      A     #Day6;  // Day 6 (Saturday)
      JNB   ED6;
      L     #EveningDay1Value;  // amount of bodies on day 1 - Evening shift (Monday)
      L     #EveningDay2Value;  // amount of bodies on day 2 - Evening shift (Tuesday)
      +I;
      L     #EveningDay3Value;  // amount of bodies on day 3 - Evening shift (Wednesday)
      +I;
      L     #EveningDay4Value;  // amount of bodies on day 4 - Evening shift (Thursday)
      +I;
      L     #EveningDay5Value;  // amount of bodies on day 5 - Evening shift (Friday)
      +I;
      L     #EveningDay6Value;  // amount of bodies on day 6 - Evening shift (Saturday)
      +I;
      T     #H_Out.TotalEvening;  // copy to HMI
ED6:  NOP   0;

      A     #Day7;  // Day 7 (Sunday)
      JNB   ED7;
      L     #EveningDay1Value;  // amount of bodies on day 1 - Evening shift (Monday)
      L     #EveningDay2Value;  // amount of bodies on day 2 - Evening shift (Tuesday)
      +I;
      L     #EveningDay3Value;  // amount of bodies on day 3 - Evening shift (Wednesday)
      +I;
      L     #EveningDay4Value;  // amount of bodies on day 4 - Evening shift (Thursday)
      +I;
      L     #EveningDay5Value;  // amount of bodies on day 5 - Evening shift (Friday)
      +I;
      L     #EveningDay6Value;  // amount of bodies on day 6 - Evening shift (Saturday)
      +I;
      L     #EveningDay7Value;  // amount of bodies on day 7 - Evening shift (Sunday)
      +I;
      T     #H_Out.TotalEvening;  // copy to HMI
ED7:  NOP   0;


NETWORK
TITLE = **** 4.4 - Machine status - Calculated **** Production value Night shift
// Production value Night shift
      A     #Day1;  // Day 1 (Monday)
      JNB   ND1;
      L     #NightDay1Value;  // amount of bodies on day 1 - Night shift (Monday)
      T     #H_Out.TotalNight;  // copy to HMI
ND1:  NOP   0;

      A     #Day2;  // Day 2 (tuesday)
      JNB   ND2;
      L     #NightDay1Value;  // amount of bodies on day 1 - Night shift (Monday)
      L     #NightDay2Value;  // amount of bodies on day 2 - Night shift (Tuesday)
      T     #H_Out.TotalNight;  // copy to HMI
ND2:  NOP   0;

      A     #Day3;  // Day 3 (Wednesday)
      JNB   ND3;
      L     #NightDay1Value;  // amount of bodies on day 1 - Night shift (Monday)
      L     #NightDay2Value;  // amount of bodies on day 2 - Night shift (Tuesday)
      +I;
      L     #NightDay3Value;  // amount of bodies on day 3 - Night shift (Wednesday)
      +I;
      T     #H_Out.TotalNight;  // copy to HMI
ND3:  NOP   0;

      A     #Day4;  // Day 4 (tuesday)
      JNB   ND4;
      L     #NightDay1Value;  // amount of bodies on day 1 - Night shift (Monday)
      L     #NightDay2Value;  // amount of bodies on day 2 - Night shift (Tuesday)
      +I;
      L     #NightDay3Value;  // amount of bodies on day 3 - Night shift (Wednesday)
      +I;
      L     #NightDay4Value;  // amount of bodies on day 4 - Night shift (Thursday)
      +I;
      T     #H_Out.TotalNight;  // copy to HMI
ND4:  NOP   0;

      A     #Day5;  // Day 5 (Friday)
      JNB   ND5;
      L     #NightDay1Value;  // amount of bodies on day 1 - Night shift (Monday)
      L     #NightDay2Value;  // amount of bodies on day 2 - Night shift (Tuesday)
      +I;
      L     #NightDay3Value;  // amount of bodies on day 3 - Night shift (Wednesday)
      +I;
      L     #NightDay4Value;  // amount of bodies on day 4 - Night shift (Thursday)
      +I;
      L     #NightDay5Value;  // amount of bodies on day 5 - Night shift (Friday)
      +I;
      T     #H_Out.TotalNight;  // copy to HMI
ND5:  NOP   0;

      A     #Day6;  // Day 6 (Saturday)
      JNB   ND6;
      L     #NightDay1Value;  // amount of bodies on day 1 - Night shift (Monday)
      L     #NightDay2Value;  // amount of bodies on day 2 - Night shift (Tuesday)
      +I;
      L     #NightDay3Value;  // amount of bodies on day 3 - Night shift (Wednesday)
      +I;
      L     #NightDay4Value;  // amount of bodies on day 4 - Night shift (Thursday)
      +I;
      L     #NightDay5Value;  // amount of bodies on day 5 - Night shift (Friday)
      +I;
      L     #NightDay6Value;  // amount of bodies on day 6 - Night shift (Saturday)
      +I;
      T     #H_Out.TotalNight;  // copy to HMI
ND6:  NOP   0;

      A     #Day7;  // Day 7 (Sunday)
      JNB   ND7;
      L     #NightDay1Value;  // amount of bodies on day 1 - Night shift (Monday)
      L     #NightDay2Value;  // amount of bodies on day 2 - Night shift (Tuesday)
      +I;
      L     #NightDay3Value;  // amount of bodies on day 3 - Night shift (Wednesday)
      +I;
      L     #NightDay4Value;  // amount of bodies on day 4 - Night shift (Thursday)
      +I;
      L     #NightDay5Value;  // amount of bodies on day 5 - Night shift (Friday)
      +I;
      L     #NightDay6Value;  // amount of bodies on day 6 - Night shift (Saturday)
      +I;
      L     #NightDay7Value;  // amount of bodies on day 7 - Evening shift (Sunday)
      +I;
      T     #H_Out.TotalNight;  // copy to HMI
ND7:  NOP   0;


NETWORK
TITLE = **** 4.4 - Machine status - Calculated **** Production value Week on day 1
// Production value Week on day 1
      A     #Day1;  // Day 1 (Monday)
      JNB   day1;
      L     #Day1Value;  // amount of bodies on day 1 (Monday)
      T     #WeekValue;  // copy to HMI
day1: NOP   0;

NETWORK
TITLE = **** 4.4 - Machine status - Calculated **** Production value Week on day 2
// Production value Week on day 2
      A     #Day2;  // Day 2 (tuesday)
      JNB   day2;
      L     #Day1Value;  // amount of bodies on day 1 (Monday)
      L     #Day2Value;  // amount of bodies on day 2 (Tuesday)
      +I;
      T     #WeekValue;  // copy to HMI
day2: NOP   0;

NETWORK
TITLE = **** 4.4 - Machine status - Calculated **** Production value Week on day 3
// Production value Week on day 3
      A     #Day3;  // Day 3 (Wednesday)
      JNB   day3;
      L     #Day1Value;  // amount of bodies on day 1 (Monday)
      L     #Day2Value;  // amount of bodies on day 2 (Tuesday)
      +I;
      L     #Day3Value;  // amount of bodies on day 3 (Wednesday)
      +I;
      T     #WeekValue;  // copy to HMI
day3: NOP   0;

NETWORK
TITLE = **** 4.4 - Machine status - Calculated **** Production value Week on day 4
// Production value Week on day 4
      A     #Day4;  // Day 4 (tuesday)
      JNB   day4;
      L     #Day1Value;  // amount of bodies on day 1 (Monday)
      L     #Day2Value;  // amount of bodies on day 2 (Tuesday)
      +I;
      L     #Day3Value;  // amount of bodies on day 3 (Wednesday)
      +I;
      L     #Day4Value;  // amount of bodies on day 4 (Thursday)
      +I;
      T     #WeekValue;  // copy to HMI
day4: NOP   0;

NETWORK
TITLE = **** 4.4 - Machine status - Calculated **** Production value Week on day 5
// Production value Week on day 5
      A     #Day5;  // Day 5 (Friday)
      JNB   day5;
      L     #Day1Value;  // amount of bodies on day 1 (Monday)
      L     #Day2Value;  // amount of bodies on day 2 (Tuesday)
      +I;
      L     #Day3Value;  // amount of bodies on day 3 (Wednesday)
      +I;
      L     #Day4Value;  // amount of bodies on day 4 (Thursday)
      +I;
      L     #Day5Value;  // amount of bodies on day 5 (Friday)
      +I;
      T     #WeekValue;  // copy to HMI
day5: NOP   0;

NETWORK
TITLE = **** 4.4 - Machine status - Calculated **** Production value Week on day 6
// Production value Week on day 6
      A     #Day6;  // Day 6 (Saturday)
      JNB   day6;
      L     #Day1Value;  // amount of bodies on day 1 (Monday)
      L     #Day2Value;  // amount of bodies on day 2 (Tuesday)
      +I;
      L     #Day3Value;  // amount of bodies on day 3 (Wednesday)
      +I;
      L     #Day4Value;  // amount of bodies on day 4 (Thursday)
      +I;
      L     #Day5Value;  // amount of bodies on day 5 (Friday)
      +I;
      L     #Day6Value;  // amount of bodies on day 6 (Saturday)
      +I;
      T     #WeekValue;  // copy to HMI
day6: NOP   0;

NETWORK
TITLE = **** 4.4 - Machine status - Calculated **** Production value Week on day 7
// Production value Week on day 7
      A     #Day7;  // Day 7 (Sunday)
      JNB   day7;
      L     #Day1Value;  // amount of bodies on day 1 (Monday)
      L     #Day2Value;  // amount of bodies on day 2 (Tuesday)
      +I;
      L     #Day3Value;  // amount of bodies on day 3 (Wednesday)
      +I;
      L     #Day4Value;  // amount of bodies on day 4 (Thursday)
      +I;
      L     #Day5Value;  // amount of bodies on day 5 (Friday)
      +I;
      L     #Day6Value;  // amount of bodies on day 6 (Saturday)
      +I;
      L     #Day7Value;  // amount of bodies on day 7 (Sunday)
      +I;
      T     #WeekValue;  // copy to HMI
day7: NOP   0;

REGION Network 39: **** 4.6 - Machine status - Indications **** Icon Animation
   // Icon Animation for HMI
   IF "TRUE" THEN
       "LSimpleIAnim"(I_SetPos := "FALSE",
                      I_ResetPos := "FALSE",
                      I_Active := "FALSE",
                      I_Invisible := "FALSE",
                      I_OutOfUse := "FALSE",
                      I_AlarmA := "FALSE",
                      I_AlarmB := "FALSE",
                      I_AlarmC := "FALSE",
                      I_AlarmD := "FALSE",
                      I_ManualMode := "FALSE",
                      I_FncSelInHMI := "FALSE",
                      H_IAnim => #H_IAnim);
   END_IF;
END_REGION

REGION Network 40: **** 4.6 - Machine status - Indications **** Animation
   // Animation
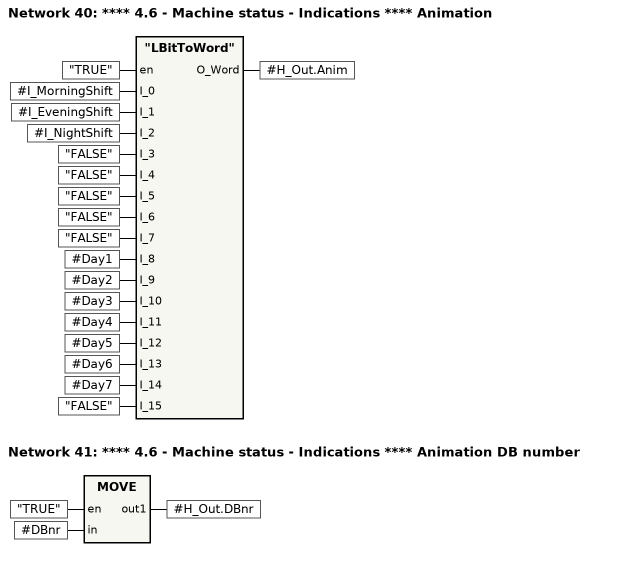
   IF "TRUE" THEN
       "LBitToWord"(I_0 := #I_MorningShift,
                    I_1 := #I_EveningShift,
                    I_2 := #I_NightShift,
                    I_3 := "FALSE",
                    I_4 := "FALSE",
                    I_5 := "FALSE",
                    I_6 := "FALSE",
                    I_7 := "FALSE",
                    I_8 := #Day1,
                    I_9 := #Day2,
                    I_10 := #Day3,
                    I_11 := #Day4,
                    I_12 := #Day5,
                    I_13 := #Day6,
                    I_14 := #Day7,
                    I_15 := "FALSE",
                    O_Word => #H_Out.Anim);
   END_IF;
END_REGION

REGION Network 41: **** 4.6 - Machine status - Indications **** Animation DB number
   // Animation DB number
   IF "TRUE" THEN #H_Out.DBnr := #DBnr; END_IF;
END_REGION

NETWORK
TITLE = **** 8 - Outputs **** Copy of counters for day activities to HMI
// Copy of counters for day activities to HMI
      L     #MorningDay1Value;  // amount of bodies on day 1 - Morning shift (Monday)
      T     #H_Out.MorningDay1Value;  // copy to HMI

      L     #EveningDay1Value;  // amount of bodies on day 1 - Evening shift (Monday)
      T     #H_Out.EveningDay1Value;  // copy to HMI

      L     #NightDay1Value;  // amount of bodies on day 1 - Night shift (Monday)
      T     #H_Out.NightDay1Value;  // copy to HMI

      L     #MorningDay2Value;  // amount of bodies on day 2 - Morning shift (Tuesday)
      T     #H_Out.MorningDay2Value;  // copy to HMI

      L     #EveningDay2Value;  // amount of bodies on day 2 - Evening shift (Tuesday)
      T     #H_Out.EveningDay2Value;  // copy to HMI

      L     #NightDay2Value;  // amount of bodies on day 2 - Night shift (Tuesday)
      T     #H_Out.NightDay2Value;  // copy to HMI

      L     #MorningDay3Value;  // amount of bodies on day 3 - Morning shift (Wednesday)
      T     #H_Out.MorningDay3Value;  // copy to HMI

      L     #EveningDay3Value;  // amount of bodies on day 3 - Evening shift (Wednesday)
      T     #H_Out.EveningDay3Value;  // copy to HMI

      L     #NightDay3Value;  // amount of bodies on day 3 - Night shift (Wednesday)
      T     #H_Out.NightDay3Value;  // copy to HMI

      L     #MorningDay4Value;  // amount of bodies on day 4 - Morning shift (Thursday)
      T     #H_Out.MorningDay4Value;  // copy to HMI

      L     #EveningDay4Value;  // amount of bodies on day 4 - Evening shift (Thursday)
      T     #H_Out.EveningDay4Value;  // copy to HMI

      L     #NightDay4Value;  // amount of bodies on day 4 - Night shift (Thursday)
      T     #H_Out.NightDay4Value;  // copy to HMI

      L     #MorningDay5Value;  // amount of bodies on day 5 - Morning shift (Friday)
      T     #H_Out.MorningDay5Value;  // copy to HMI

      L     #EveningDay5Value;  // amount of bodies on day 5 - Evening shift (Friday)
      T     #H_Out.EveningDay5Value;  // copy to HMI

      L     #NightDay5Value;  // amount of bodies on day 5 - night shift (Friday)
      T     #H_Out.NightDay5Value;  // copy to HMI

      L     #MorningDay6Value;  // amount of bodies on day 6 - Morning shift (Saturday)
      T     #H_Out.MorningDay6Value;  // copy to HMI

      L     #EveningDay6Value;  // amount of bodies on day 6 - Evening shift (Saturday)
      T     #H_Out.EveningDay6Value;  // copy to HMI

      L     #NightDay6Value;  // amount of bodies on day 6 - Night shift (Saturday)
      T     #H_Out.NightDay6Value;  // copy to HMI

      L     #MorningDay7Value;  // amount of bodies on day 7 - Morning shift (Sunday)
      T     #H_Out.MorningDay7Value;  // copy to HMI

      L     #EveningDay7Value;  // amount of bodies on day 7 - Evening shift (Sunday)
      T     #H_Out.EveningDay7Value;  // copy to HMI

      L     #NightDay7Value;  // amount of bodies on day 7 - Night shift (Sunday)
      T     #H_Out.NightDay7Value;  // copy to HMI

NETWORK
TITLE = **** 8 - Outputs **** Copy of counters for summation per day to HMI
// Copy of counters for summation per day to HMI
      L     #Day1Value;  // amount of bodies on day 1 (Monday)
      T     #H_Out.Day1Value;  // copy to HMI

      L     #Day2Value;  // amount of bodies on day 2 (Tuesday)
      T     #H_Out.Day2Value;  // copy to HMI

      L     #Day3Value;  // amount of bodies on day 3 (Wednesday)
      T     #H_Out.Day3Value;  // copy to HMI

      L     #Day4Value;  // amount of bodies on day 4 (Thursday)
      T     #H_Out.Day4Value;  // copy to HMI

      L     #Day5Value;  // amount of bodies on day 5 (Friday)
      T     #H_Out.Day5Value;  // copy to HMI

      L     #Day6Value;  // amount of bodies on day 6 (Saturday)
      T     #H_Out.Day6Value;  // copy to HMI

      L     #Day7Value;  // amount of bodies on day 7 (Sunday)
      T     #H_Out.Day7Value;  // copy to HMI

NETWORK
TITLE = **** 8 - Outputs **** Copy of counter for the complete week to HMI
// Copy of counter for the complete week to HMI
      L     #WeekValue;  // amount of bodies during week
      T     #H_Out.WeekValue;  // copy to HMI

NETWORK
TITLE = **** 8 - Outputs **** Copy of global counter to HMI
// Copy of global counter to HMI
      L     #TotalValue;  // amount of bodies
      T     #H_Out.TotalValue;  // copy to HMI
END_FUNCTION_BLOCK

FUNCTION_BLOCK "LDP/PNCouplerCheck"   // FB1900, FBD
TITLE = LDPCouplerCheck
{ S7_Optimized_Access := 'FALSE' }
AUTHOR : VCC
FAMILY : Communic
NAME : LDPCheck
VERSION : 0.1
// ================================================================================
// This FB checks the communication between 2 plc's via DP/DP coupler
// ================================================================================
// stored: AutoNumber false, IsIECCheckEnabled false, SetENOAutomatically False, UDAEnableTagReadback false
   VAR_INPUT
      I_CheckPlcCom { ExternalAccessible := 'False'; ExternalVisible := 'False'; ExternalWritable := 'False'} : Bool;   // Input from other plc via DP/DP coupler
      I_AlarmResetPB { ExternalAccessible := 'False'; ExternalVisible := 'False'; ExternalWritable := 'False'} : Bool;   // Alarm reset pushbutton is activated
   END_VAR
   VAR_OUTPUT
      O_CheckPlcCom { ExternalAccessible := 'False'; ExternalVisible := 'False'; ExternalWritable := 'False'} : Bool;   // Output to other plc via DP/DP coupler
      O_DPCouplerResponseAlarm { ExternalAccessible := 'False'; ExternalVisible := 'False'; ExternalWritable := 'False'} : Bool;   // Profibus DP coupler alarm
      O_AlarmABCondition { ExternalAccessible := 'False'; ExternalVisible := 'False'; ExternalWritable := 'False'} : Bool;   // Alarm AB condition
      H_IAnim { ExternalAccessible := 'False'; ExternalVisible := 'False'; ExternalWritable := 'False'} : Word;   // Animation
   END_VAR
   VAR DB_SPECIFIC
      H_Out : Struct   // HMI
         Anim : Word;   // HMI Animation of the object
         DBnr : Int;   // HMI Animation DB number
      END_STRUCT;
      DPCouplerResponseAlarm { ExternalAccessible := 'False'; ExternalVisible := 'False'; ExternalWritable := 'False'} : Bool;   // Profibus DP coupler alarm
      ResponseTimeOffAlarm { ExternalAccessible := 'False'; ExternalVisible := 'False'; ExternalWritable := 'False'} : Bool;   // Alarm : signal from other plc stays ON
      ResponseTimeOnAlarm { ExternalAccessible := 'False'; ExternalVisible := 'False'; ExternalWritable := 'False'} : Bool;   // Alarm : signal from other plc stays OFF
      ChangeStatePulse { ExternalAccessible := 'False'; ExternalVisible := 'False'; ExternalWritable := 'False'} : Bool;   // Pulse to change state every 3 sec
      CheckPLC { ExternalAccessible := 'False'; ExternalVisible := 'False'; ExternalWritable := 'False'} : Bool;   // Variable changing from state every 3 sec
      CheckPlcCom { ExternalAccessible := 'False'; ExternalVisible := 'False'; ExternalWritable := 'False'} : Bool;   // Variable changing from state every 3 sec
      ChangeStateTime { ExternalAccessible := 'False'; ExternalVisible := 'False'; ExternalWritable := 'False'} : DInt := DINT#3000;   // Time between 2 pulses
      AlarmResponseTime { ExternalAccessible := 'False'; ExternalVisible := 'False'; ExternalWritable := 'False'} : DInt := DINT#5000;   // Time to create alarm
      DPCouplerResponseAlmCond { ExternalAccessible := 'False'; ExternalVisible := 'False'; ExternalWritable := 'False'} : Bool;   // Profibus DP coupler alarm condition
      DBnr { ExternalAccessible := 'False'; ExternalVisible := 'False'; ExternalWritable := 'False'} : Int;   // HMI DB number
      InputCheckPlcCom { ExternalAccessible := 'False'; ExternalVisible := 'False'; ExternalWritable := 'False'} : Bool;   // Input from other plc via DP/DP coupler
   END_VAR
   VAR
      ResponsTimer1 { ExternalAccessible := 'False'; ExternalVisible := 'False'; ExternalWritable := 'False'; S7_SetPoint := 'True'} : "LTimer";   // Timer to create alarm
      ResponsTimer2 { ExternalAccessible := 'False'; ExternalVisible := 'False'; ExternalWritable := 'False'; S7_SetPoint := 'True'} : "LTimer";   // Timer to create alarm
      StateTimer { ExternalAccessible := 'False'; ExternalVisible := 'False'; ExternalWritable := 'False'; S7_SetPoint := 'True'} : "LTimer";   // Timer to create pulse to change status
   END_VAR
BEGIN

NETWORK
TITLE = **** 1 - Inputs **** DB number
// DB number
      L     DINO;
      T     #DBnr;

REGION Network 2: **** 1 - Inputs **** Input from other plc via DP/DP coupler
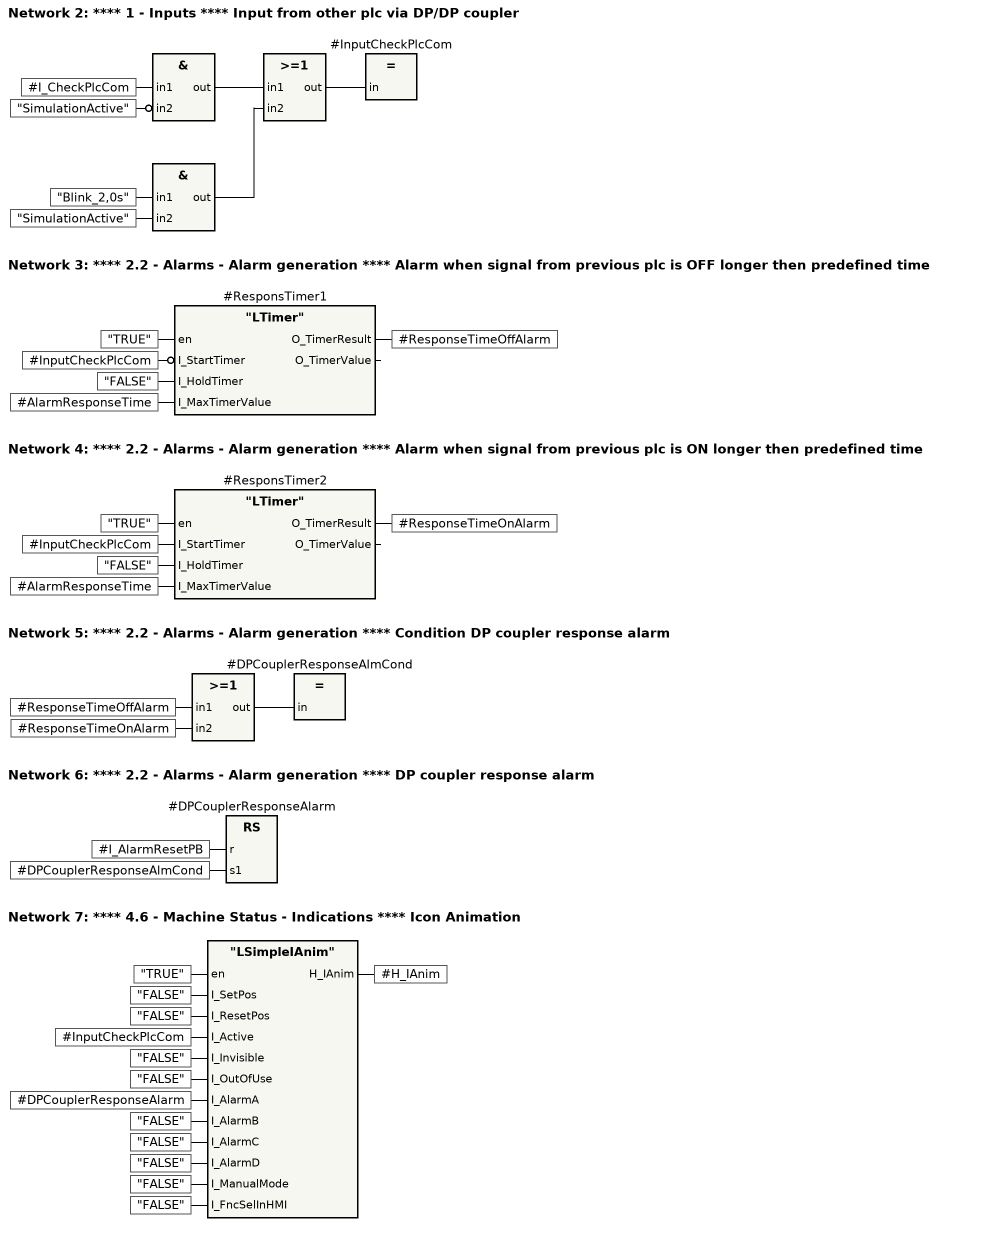
   #InputCheckPlcCom := (#I_CheckPlcCom AND NOT "SimulationActive") OR ("Blink_2,0s" AND "SimulationActive");
END_REGION

REGION Network 3: **** 2.2 - Alarms - Alarm generation **** Alarm when signal from previous plc is OFF longer then predefined time
   // Alarm when signal from previous plc is OFF longer then predefined time
   IF "TRUE" THEN
       #ResponsTimer1(I_StartTimer := NOT #InputCheckPlcCom,   // "LTimer"
                      I_HoldTimer := "FALSE",
                      I_MaxTimerValue := #AlarmResponseTime,
                      O_TimerResult => #ResponseTimeOffAlarm);
   END_IF;
END_REGION

REGION Network 4: **** 2.2 - Alarms - Alarm generation **** Alarm when signal from previous plc is ON longer then predefined time
   // Alarm when signal from previous plc is ON longer then predefined time
   IF "TRUE" THEN
       #ResponsTimer2(I_StartTimer := #InputCheckPlcCom,   // "LTimer"
                      I_HoldTimer := "FALSE",
                      I_MaxTimerValue := #AlarmResponseTime,
                      O_TimerResult => #ResponseTimeOnAlarm);
   END_IF;
END_REGION

REGION Network 5: **** 2.2 - Alarms - Alarm generation **** Condition DP coupler response alarm
   // Condition DP coupler response alarm
   #DPCouplerResponseAlmCond := #ResponseTimeOffAlarm OR #ResponseTimeOnAlarm;
END_REGION

REGION Network 6: **** 2.2 - Alarms - Alarm generation **** DP coupler response alarm
   // DP coupler response alarm
   IF #I_AlarmResetPB THEN
       #DPCouplerResponseAlarm := FALSE;   // RS flip-flop
   END_IF;
   IF #DPCouplerResponseAlmCond THEN #DPCouplerResponseAlarm := TRUE; END_IF;
END_REGION

REGION Network 7: **** 4.6 - Machine Status - Indications **** Icon Animation
   // Icon Animation
   IF "TRUE" THEN
       "LSimpleIAnim"(I_SetPos := "FALSE",
                      I_ResetPos := "FALSE",
                      I_Active := #InputCheckPlcCom,
                      I_Invisible := "FALSE",
                      I_OutOfUse := "FALSE",
                      I_AlarmA := #DPCouplerResponseAlarm,
                      I_AlarmB := "FALSE",
                      I_AlarmC := "FALSE",
                      I_AlarmD := "FALSE",
                      I_ManualMode := "FALSE",
                      I_FncSelInHMI := "FALSE",
                      H_IAnim => #H_IAnim);
   END_IF;
END_REGION

REGION Network 8: **** 4.6 - Machine Status - Indications **** Animation
   // Animation
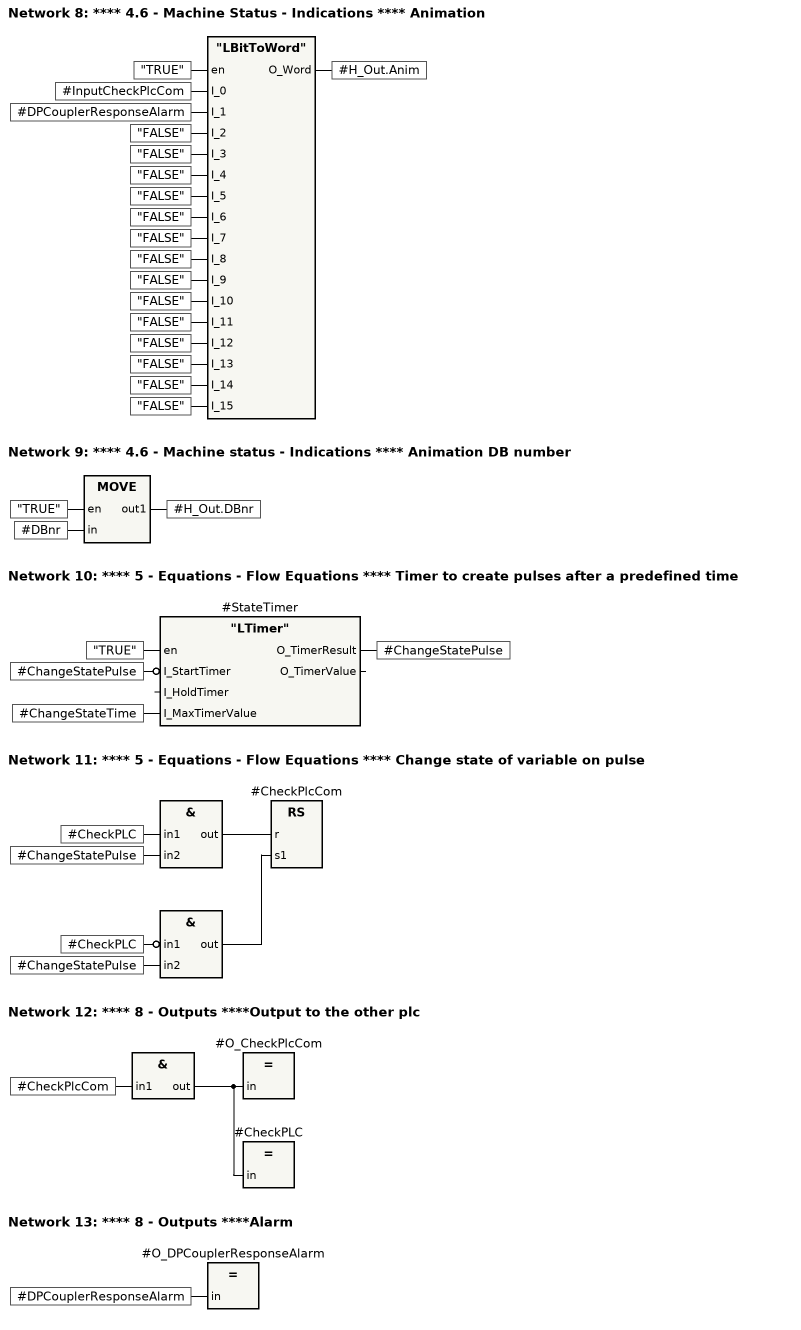
   IF "TRUE" THEN
       "LBitToWord"(I_0 := #InputCheckPlcCom,
                    I_1 := #DPCouplerResponseAlarm,
                    I_2 := "FALSE",
                    I_3 := "FALSE",
                    I_4 := "FALSE",
                    I_5 := "FALSE",
                    I_6 := "FALSE",
                    I_7 := "FALSE",
                    I_8 := "FALSE",
                    I_9 := "FALSE",
                    I_10 := "FALSE",
                    I_11 := "FALSE",
                    I_12 := "FALSE",
                    I_13 := "FALSE",
                    I_14 := "FALSE",
                    I_15 := "FALSE",
                    O_Word => #H_Out.Anim);
   END_IF;
END_REGION

REGION Network 9: **** 4.6 - Machine status - Indications **** Animation DB number
   // Animation DB number
   IF "TRUE" THEN #H_Out.DBnr := #DBnr; END_IF;
END_REGION

REGION Network 10: **** 5 - Equations - Flow Equations **** Timer to create pulses after a predefined time
   // Timer to create pulses after a predefined time
   IF "TRUE" THEN
       #StateTimer(I_StartTimer := NOT #ChangeStatePulse,   // "LTimer"
                   I_MaxTimerValue := #ChangeStateTime,
                   O_TimerResult => #ChangeStatePulse);
   END_IF;
END_REGION

REGION Network 11: **** 5 - Equations - Flow Equations **** Change state of variable on pulse
   // Change state of variable on pulse
   IF #CheckPLC AND #ChangeStatePulse THEN
       #CheckPlcCom := FALSE;   // RS flip-flop
   END_IF;
   IF NOT #CheckPLC AND #ChangeStatePulse THEN #CheckPlcCom := TRUE; END_IF;
END_REGION

REGION Network 12: **** 8 - Outputs ****Output to the other plc
   // Output to the other plc
   #O_CheckPlcCom := #CheckPlcCom;
   #CheckPLC := #CheckPlcCom;
END_REGION

REGION Network 13: **** 8 - Outputs ****Alarm
   // Alarm
   #O_DPCouplerResponseAlarm := #DPCouplerResponseAlarm;
END_REGION

REGION Network 14: **** 8 - Outputs **** Alarm Resetable
   // Alarm Resetable
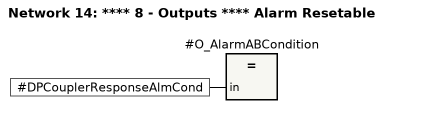
   #O_AlarmABCondition := #DPCouplerResponseAlmCond;
END_REGION
END_FUNCTION_BLOCK

FUNCTION_BLOCK "LDP/PNCouplerDiag"   // FB1901, FBD
TITLE = LDPCouplerDiag
{ S7_Optimized_Access := 'FALSE' }
AUTHOR : VCC
FAMILY : Communic
NAME : LDPDiag
VERSION : 0.1
// ================================================================================
// Function used to read the diagnostic information from a DP/DP coupler.
// ================================================================================
// stored: AutoNumber false, IsIECCheckEnabled false, SetENOAutomatically False, UDAEnableTagReadback false
   VAR_INPUT
      I_PNPNSendError { ExternalAccessible := 'False'; ExternalVisible := 'False'; ExternalWritable := 'False'} : Bool;   // Send Error
      I_PNPNSendSUBSOn { ExternalAccessible := 'False'; ExternalVisible := 'False'; ExternalWritable := 'False'} : Bool;   // SUBS ON
      I_PNPNDiagSend { ExternalAccessible := 'False'; ExternalVisible := 'False'; ExternalWritable := 'False'} : Byte;   // Diag
      I_PNPNRcvError { ExternalAccessible := 'False'; ExternalVisible := 'False'; ExternalWritable := 'False'} : Bool;   // Recv Error
      I_PNPNRcvSUBSOn { ExternalAccessible := 'False'; ExternalVisible := 'False'; ExternalWritable := 'False'} : Bool;   // SUBS ON
      I_PNPNRcvAckReq { ExternalAccessible := 'False'; ExternalVisible := 'False'; ExternalWritable := 'False'} : Bool;   // ACK REQ
      I_PNPNDiagRecv { ExternalAccessible := 'False'; ExternalVisible := 'False'; ExternalWritable := 'False'} : Byte;   // Diag
      I_AlarmResetPB { ExternalAccessible := 'False'; ExternalVisible := 'False'; ExternalWritable := 'False'} : Bool;   // Alarm reset pushbutton is activated
   END_VAR
   VAR_OUTPUT
      O_Alarm { ExternalAccessible := 'False'; ExternalVisible := 'False'; ExternalWritable := 'False'} : Bool;   // Alarm
      O_AlarmABCondition { ExternalAccessible := 'False'; ExternalVisible := 'False'; ExternalWritable := 'False'} : Bool;   // Alarms AB condition
      H_IAnim { ExternalAccessible := 'False'; ExternalVisible := 'False'; ExternalWritable := 'False'} : Word;   // Icon Animation
   END_VAR
   VAR DB_SPECIFIC
      H_Out : Struct   // HMI
         Anim : Word;   // HMI Animation of the object
         DBnr : Int;   // HMI Animation DB number
      END_STRUCT;
      Alarm { ExternalAccessible := 'False'; ExternalVisible := 'False'; ExternalWritable := 'False'} : Bool;   // Alarm
      Send_error { ExternalAccessible := 'False'; ExternalVisible := 'False'; ExternalWritable := 'False'} : Bool;   // Send Error
      Send_SubOn { ExternalAccessible := 'False'; ExternalVisible := 'False'; ExternalWritable := 'False'} : Bool;   // Send sub on
      Send_TimeOut { ExternalAccessible := 'False'; ExternalVisible := 'False'; ExternalWritable := 'False'} : Bool;   // Send time out
      Send_SeqNrError { ExternalAccessible := 'False'; ExternalVisible := 'False'; ExternalWritable := 'False'} : Bool;   // Send sequenz number error
      Send_CRCError { ExternalAccessible := 'False'; ExternalVisible := 'False'; ExternalWritable := 'False'} : Bool;   // Send CRC error
      Receive_Error { ExternalAccessible := 'False'; ExternalVisible := 'False'; ExternalWritable := 'False'} : Bool;   // Receive error
      Receive_SubOn { ExternalAccessible := 'False'; ExternalVisible := 'False'; ExternalWritable := 'False'} : Bool;   // Receive sub on
      Receive_AckReq { ExternalAccessible := 'False'; ExternalVisible := 'False'; ExternalWritable := 'False'} : Bool;   // Reveice ack request
      Receive_TimeOut { ExternalAccessible := 'False'; ExternalVisible := 'False'; ExternalWritable := 'False'} : Bool;   // Receive time out
      Receive_SeqNrError { ExternalAccessible := 'False'; ExternalVisible := 'False'; ExternalWritable := 'False'} : Bool;   // Receive sequenz number error
      Receive_CRCError { ExternalAccessible := 'False'; ExternalVisible := 'False'; ExternalWritable := 'False'} : Bool;   // Receive CRC error
      AlarmCond { ExternalAccessible := 'False'; ExternalVisible := 'False'; ExternalWritable := 'False'} : Bool;   // Alarm condition
      DBnr { ExternalAccessible := 'False'; ExternalVisible := 'False'; ExternalWritable := 'False'} : Int;   // HMI DB number
   END_VAR
BEGIN

NETWORK
TITLE = **** 1 - Inputs **** DB number
// DB number
      L     DINO;
      T     #DBnr;

REGION Network 2: **** 1 - Inputs **** Information SEND
   // Information SEND
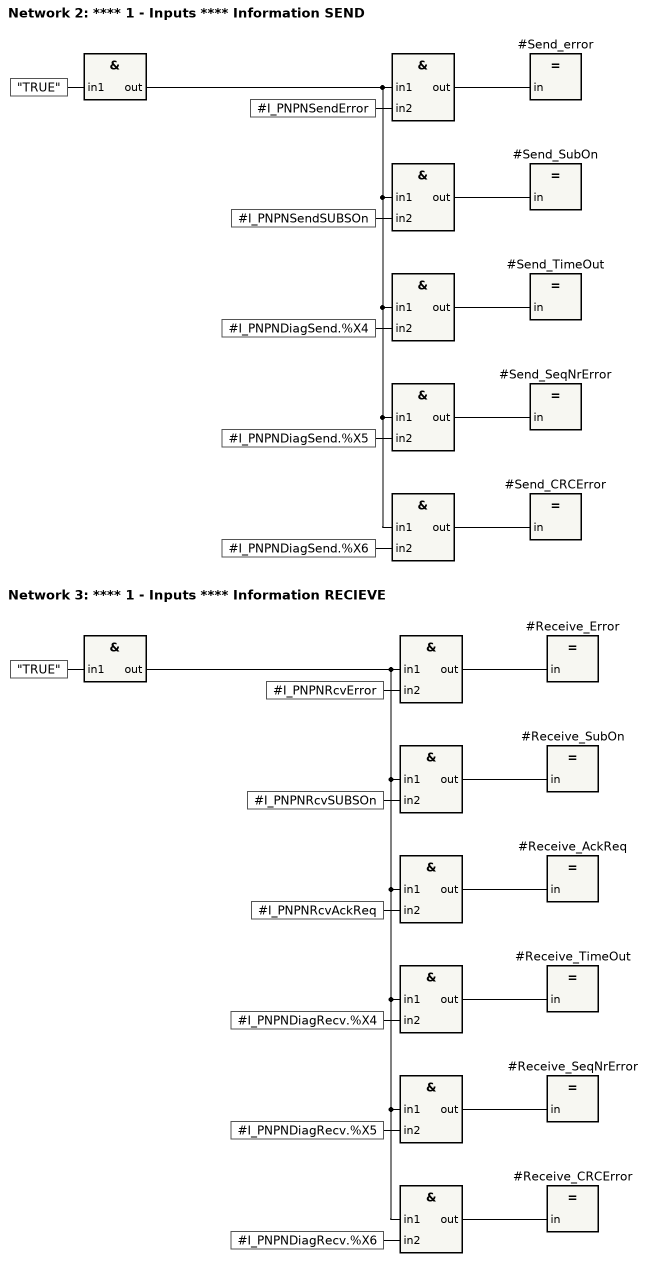
   #Send_error := "TRUE" AND #I_PNPNSendError;
   #Send_SubOn := "TRUE" AND #I_PNPNSendSUBSOn;
   #Send_TimeOut := "TRUE" AND #I_PNPNDiagSend.%X4;
   #Send_SeqNrError := "TRUE" AND #I_PNPNDiagSend.%X5;
   #Send_CRCError := "TRUE" AND #I_PNPNDiagSend.%X6;
END_REGION

REGION Network 3: **** 1 - Inputs **** Information RECIEVE
   // Information RECIEVE
   #Receive_Error := "TRUE" AND #I_PNPNRcvError;
   #Receive_SubOn := "TRUE" AND #I_PNPNRcvSUBSOn;
   #Receive_AckReq := "TRUE" AND #I_PNPNRcvAckReq;
   #Receive_TimeOut := "TRUE" AND #I_PNPNDiagRecv.%X4;
   #Receive_SeqNrError := "TRUE" AND #I_PNPNDiagRecv.%X5;
   #Receive_CRCError := "TRUE" AND #I_PNPNDiagRecv.%X6;
END_REGION

REGION Network 4: **** 2.2 - Alarms - Alarm generation **** Condition send/Recive alarm
   // Condition send/Recive alarm
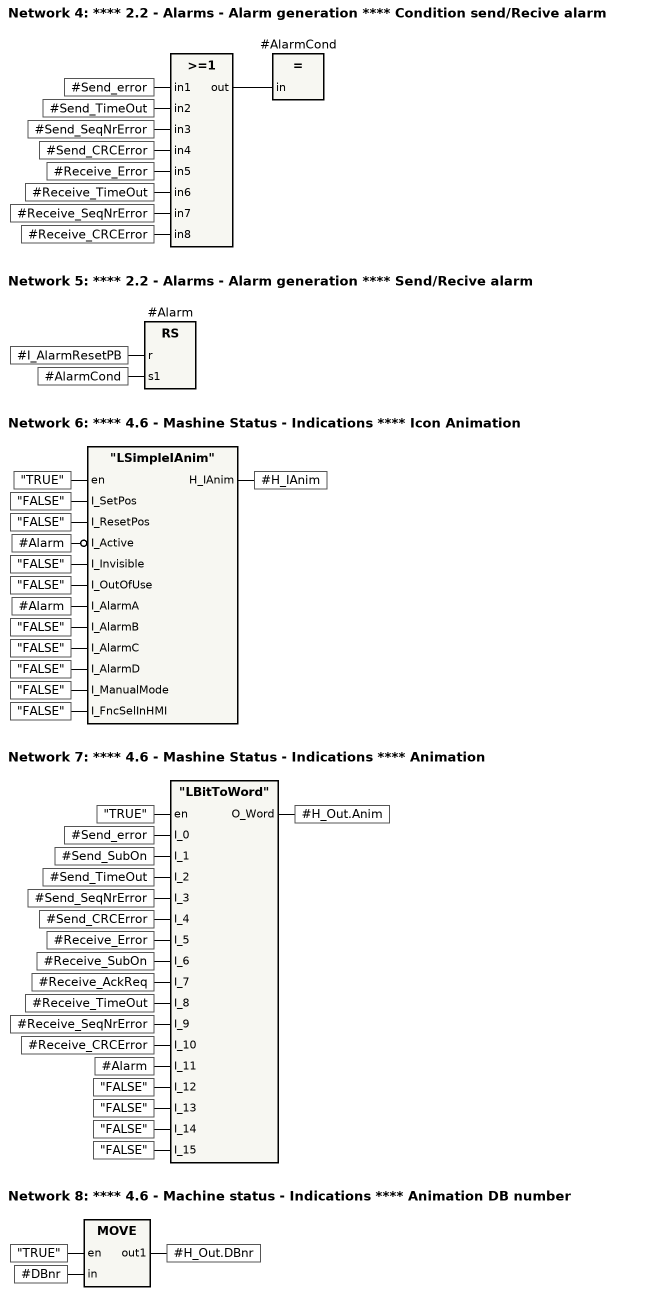
   #AlarmCond := #Send_error OR #Send_TimeOut OR #Send_SeqNrError OR #Send_CRCError OR #Receive_Error OR #Receive_TimeOut OR #Receive_SeqNrError OR #Receive_CRCError;
END_REGION

REGION Network 5: **** 2.2 - Alarms - Alarm generation **** Send/Recive alarm
   // Send/Recive alarm
   IF #I_AlarmResetPB THEN
       #Alarm := FALSE;   // RS flip-flop
   END_IF;
   IF #AlarmCond THEN #Alarm := TRUE; END_IF;
END_REGION

REGION Network 6: **** 4.6 - Mashine Status - Indications **** Icon Animation
   // Icon Animation
   IF "TRUE" THEN
       "LSimpleIAnim"(I_SetPos := "FALSE",
                      I_ResetPos := "FALSE",
                      I_Active := NOT #Alarm,
                      I_Invisible := "FALSE",
                      I_OutOfUse := "FALSE",
                      I_AlarmA := #Alarm,
                      I_AlarmB := "FALSE",
                      I_AlarmC := "FALSE",
                      I_AlarmD := "FALSE",
                      I_ManualMode := "FALSE",
                      I_FncSelInHMI := "FALSE",
                      H_IAnim => #H_IAnim);
   END_IF;
END_REGION

REGION Network 7: **** 4.6 - Mashine Status - Indications **** Animation
   // Animation
   IF "TRUE" THEN
       "LBitToWord"(I_0 := #Send_error,
                    I_1 := #Send_SubOn,
                    I_2 := #Send_TimeOut,
                    I_3 := #Send_SeqNrError,
                    I_4 := #Send_CRCError,
                    I_5 := #Receive_Error,
                    I_6 := #Receive_SubOn,
                    I_7 := #Receive_AckReq,
                    I_8 := #Receive_TimeOut,
                    I_9 := #Receive_SeqNrError,
                    I_10 := #Receive_CRCError,
                    I_11 := #Alarm,
                    I_12 := "FALSE",
                    I_13 := "FALSE",
                    I_14 := "FALSE",
                    I_15 := "FALSE",
                    O_Word => #H_Out.Anim);
   END_IF;
END_REGION

REGION Network 8: **** 4.6 - Machine status - Indications **** Animation DB number
   // Animation DB number
   IF "TRUE" THEN #H_Out.DBnr := #DBnr; END_IF;
END_REGION

REGION Network 9: **** 8 - Outputs **** Alarm
   // Alarm
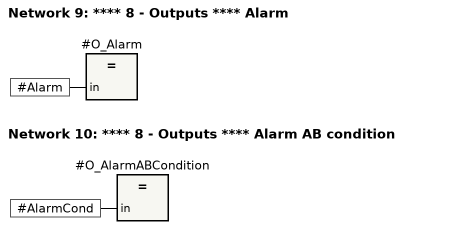
   #O_Alarm := #Alarm;
END_REGION

REGION Network 10: **** 8 - Outputs **** Alarm AB condition
   // Alarm AB condition
   #O_AlarmABCondition := #AlarmCond;
END_REGION
END_FUNCTION_BLOCK

FUNCTION_BLOCK "LChangeOfState"   // FB2103, FBD
TITLE = LChangeOfState
{ S7_Optimized_Access := 'TRUE' }
AUTHOR : VCC
FAMILY : Function
VERSION : 0.1
// =============================================================================
// This Module Handles Change Of State
// ============================================================================
// stored: AutoNumber false, IsIECCheckEnabled false, IsRetainMemResEnabled false, MemoryReserve 100, SetENOAutomatically False, UDAEnableTagReadback false
   VAR_INPUT
      I_In { ExternalAccessible := 'False'; ExternalVisible := 'False'; ExternalWritable := 'False'} : Bool;   // Input
   END_VAR
   VAR_OUTPUT
      O_OutPut { ExternalAccessible := 'False'; ExternalVisible := 'False'; ExternalWritable := 'False'} : Bool;   // Output
   END_VAR
   VAR
      PosEdge { ExternalAccessible := 'False'; ExternalVisible := 'False'; ExternalWritable := 'False'} : Bool;   // Edge
      PosEdgeResult { ExternalAccessible := 'False'; ExternalVisible := 'False'; ExternalWritable := 'False'} : Bool;   // Result
      NegEdge { ExternalAccessible := 'False'; ExternalVisible := 'False'; ExternalWritable := 'False'} : Bool;   // Edge
      NegEdgeResult { ExternalAccessible := 'False'; ExternalVisible := 'False'; ExternalWritable := 'False'} : Bool;   // Result
   END_VAR
   VAR_TEMP   // added for the SCL form of the ladder/FBD networks
      _w1 : Bool;
      _w2 : Bool;
   END_VAR
BEGIN

REGION Network 1: **** 4.4 - Machine Status - Calculation **** Create Edge
   // Create Edge
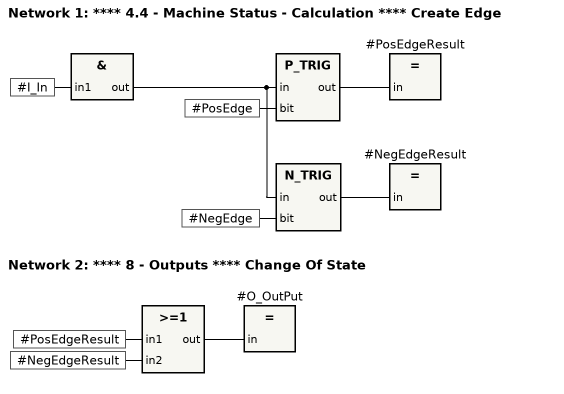
   #_w1 := #I_In AND NOT #PosEdge;   // rising edge
   #PosEdge := #I_In;
   #PosEdgeResult := #_w1;
   #_w2 := NOT #I_In AND #NegEdge;   // falling edge
   #NegEdge := #I_In;
   #NegEdgeResult := #_w2;
END_REGION

REGION Network 2: **** 8 - Outputs **** Change Of State
   // Change Of State
   #O_OutPut := #PosEdgeResult OR #NegEdgeResult;
END_REGION
END_FUNCTION_BLOCK

FUNCTION_BLOCK "LComAlarm"   // FB2105, FBD
TITLE = LComAlarm
{ S7_Optimized_Access := 'FALSE' }
AUTHOR : VCC
FAMILY : Communic
VERSION : 0.1
// =============================================================================
// This module Handles All Alarm Report To MES/VD
// =============================================================================
// stored: AutoNumber false, IsIECCheckEnabled false, SetENOAutomatically False, UDAEnableTagReadback false
   VAR_INPUT
      C_VDCommRecvDB { ExternalAccessible := 'False'; ExternalVisible := 'False'; ExternalWritable := 'False'} : DB_ANY;   // VD communication system receive DB; Not to be used by application / VD communication system receive DB; Not to be used by Application
      C_VDCommSendDB { ExternalAccessible := 'False'; ExternalVisible := 'False'; ExternalWritable := 'False'} : DB_ANY;   // VD communication system send DB; Not to be used by application / VD communication system send DB; Not to be used by Application
      C_LocalRecvDB { ExternalAccessible := 'False'; ExternalVisible := 'False'; ExternalWritable := 'False'} : DB_ANY;   // Local DB to store received data; to used by application / Local DB For Recv Data Used By The Application
      C_LocalSendDB { ExternalAccessible := 'False'; ExternalVisible := 'False'; ExternalWritable := 'False'} : DB_ANY;   // Local DB for send data; to be used by application / Local DB For Send Data Used By The Application
      C_GenAlarmDB { ExternalAccessible := 'False'; ExternalVisible := 'False'; ExternalWritable := 'False'} : DB_ANY;   // Alarm DB
      C_AlarmDBMZ1 { ExternalAccessible := 'False'; ExternalVisible := 'False'; ExternalWritable := 'False'} : DB_ANY;   // Alarm DB
      C_AlarmDBMZ2 { ExternalAccessible := 'False'; ExternalVisible := 'False'; ExternalWritable := 'False'} : DB_ANY;   // Alarm DB
      C_AlarmDBMZ3 { ExternalAccessible := 'False'; ExternalVisible := 'False'; ExternalWritable := 'False'} : DB_ANY;   // Alarm DB
      C_AlarmDBMZ4 { ExternalAccessible := 'False'; ExternalVisible := 'False'; ExternalWritable := 'False'} : DB_ANY;   // Alarm DB
      C_AlarmDBMZ5 { ExternalAccessible := 'False'; ExternalVisible := 'False'; ExternalWritable := 'False'} : DB_ANY;   // Alarm DB
      C_AlarmDBMZ6 { ExternalAccessible := 'False'; ExternalVisible := 'False'; ExternalWritable := 'False'} : DB_ANY;   // Alarm DB
      C_AlarmDBMZ7 { ExternalAccessible := 'False'; ExternalVisible := 'False'; ExternalWritable := 'False'} : DB_ANY;   // Alarm DB
      C_AlarmDBMZ8 { ExternalAccessible := 'False'; ExternalVisible := 'False'; ExternalWritable := 'False'} : DB_ANY;   // Alarm DB
      C_AlarmDBMZ9 { ExternalAccessible := 'False'; ExternalVisible := 'False'; ExternalWritable := 'False'} : DB_ANY;   // Alarm DB
      C_AlarmDBMZ10 { ExternalAccessible := 'False'; ExternalVisible := 'False'; ExternalWritable := 'False'} : DB_ANY;   // Alarm DB
      C_AlarmDBMZ11 { ExternalAccessible := 'False'; ExternalVisible := 'False'; ExternalWritable := 'False'} : DB_ANY;   // Alarm DB
      C_AlarmDBMZ12 { ExternalAccessible := 'False'; ExternalVisible := 'False'; ExternalWritable := 'False'} : DB_ANY;   // Alarm DB
      C_AlarmDBMZ13 { ExternalAccessible := 'False'; ExternalVisible := 'False'; ExternalWritable := 'False'} : DB_ANY;   // Alarm DB
      C_AlarmDBMZ14 { ExternalAccessible := 'False'; ExternalVisible := 'False'; ExternalWritable := 'False'} : DB_ANY;   // Alarm DB
      C_GenAlarmCompare { ExternalAccessible := 'False'; ExternalVisible := 'False'; ExternalWritable := 'False'} : DB_ANY;   // Alarm DB
      C_AlarmCompareDBMZ1 { ExternalAccessible := 'False'; ExternalVisible := 'False'; ExternalWritable := 'False'} : DB_ANY;   // Alarm DB
      C_AlarmCompareDBMZ2 { ExternalAccessible := 'False'; ExternalVisible := 'False'; ExternalWritable := 'False'} : DB_ANY;   // Alarm DB
      C_AlarmCompareDBMZ3 { ExternalAccessible := 'False'; ExternalVisible := 'False'; ExternalWritable := 'False'} : DB_ANY;   // Alarm DB
      C_AlarmCompareDBMZ4 { ExternalAccessible := 'False'; ExternalVisible := 'False'; ExternalWritable := 'False'} : DB_ANY;   // Alarm DB
      C_AlarmCompareDBMZ5 { ExternalAccessible := 'False'; ExternalVisible := 'False'; ExternalWritable := 'False'} : DB_ANY;   // Alarm DB
      C_AlarmCompareDBMZ6 { ExternalAccessible := 'False'; ExternalVisible := 'False'; ExternalWritable := 'False'} : DB_ANY;   // Alarm DB
      C_AlarmCompareDBMZ7 { ExternalAccessible := 'False'; ExternalVisible := 'False'; ExternalWritable := 'False'} : DB_ANY;   // Alarm DB
      C_AlarmCompareDBMZ8 { ExternalAccessible := 'False'; ExternalVisible := 'False'; ExternalWritable := 'False'} : DB_ANY;   // Alarm DB
      C_AlarmCompareDBMZ9 { ExternalAccessible := 'False'; ExternalVisible := 'False'; ExternalWritable := 'False'} : DB_ANY;   // Alarm DB
      C_AlarmCompareDBMZ10 { ExternalAccessible := 'False'; ExternalVisible := 'False'; ExternalWritable := 'False'} : DB_ANY;   // Alarm DB
      C_AlarmCompareDBMZ11 { ExternalAccessible := 'False'; ExternalVisible := 'False'; ExternalWritable := 'False'} : DB_ANY;   // Alarm DB
      C_AlarmCompareDBMZ12 { ExternalAccessible := 'False'; ExternalVisible := 'False'; ExternalWritable := 'False'} : DB_ANY;   // Alarm DB
      C_AlarmCompareDBMZ13 { ExternalAccessible := 'False'; ExternalVisible := 'False'; ExternalWritable := 'False'} : DB_ANY;   // Alarm DB
      C_AlarmCompareDBMZ14 { ExternalAccessible := 'False'; ExternalVisible := 'False'; ExternalWritable := 'False'} : DB_ANY;   // Alarm DB
      C_SubSystem { ExternalAccessible := 'False'; ExternalVisible := 'False'; ExternalWritable := 'False'} : Int;   // Number to identify the subsystem / Identify Subsystem
      C_SendDelay { ExternalAccessible := 'False'; ExternalVisible := 'False'; ExternalWritable := 'False'} : DInt;   // Send Alarm Delay
      C_NbrOfModeZone { ExternalAccessible := 'False'; ExternalVisible := 'False'; ExternalWritable := 'False'} : Int;   // Nbr Of ModeZones
      C_Filter { ExternalAccessible := 'False'; ExternalVisible := 'False'; ExternalWritable := 'False'} : Time := T#500ms;   // Filter
   END_VAR
   VAR_IN_OUT
      IO_VD : "VDComm";   // VD Comm
      IO_AlarmDB : "AlarmDB";   // Alarm
   END_VAR
   VAR
      _LVDComSubSystem { ExternalAccessible := 'False'; ExternalVisible := 'False'; ExternalWritable := 'False'; S7_SetPoint := 'True'} : "LVDComSubSystemS7-1500";   // VD Sub System Alarm
   END_VAR
   VAR DB_SPECIFIC
      ReqSendToVDAlarm { ExternalAccessible := 'False'; ExternalVisible := 'False'; ExternalWritable := 'False'} : Array[1..32] of Bool;   // Req VD
      SendAlarm { ExternalAccessible := 'False'; ExternalVisible := 'False'; ExternalWritable := 'False'} : Array[1..64] of Bool;   // Req Send Alarm
      SendAlarmDone { ExternalAccessible := 'False'; ExternalVisible := 'False'; ExternalWritable := 'False'} : Array[1..64] of Bool;   // Change Of State
      ActiveRequest { ExternalAccessible := 'False'; ExternalVisible := 'False'; ExternalWritable := 'False'} : DWord;   // No Requests Active
      OkToRequest { ExternalAccessible := 'False'; ExternalVisible := 'False'; ExternalWritable := 'False'} : Bool;   // Ok To Request New Alarm To VD
      SendDoneVD { ExternalAccessible := 'False'; ExternalVisible := 'False'; ExternalWritable := 'False'} : Bool;   // Request Is Finished
      SendToVD { ExternalAccessible := 'False'; ExternalVisible := 'False'; ExternalWritable := 'False'} : Bool;   // Send To VD
      InitUDT { ExternalAccessible := 'False'; ExternalVisible := 'False'; ExternalWritable := 'False'} : Bool;   // Init
      DelaySend { ExternalAccessible := 'False'; ExternalVisible := 'False'; ExternalWritable := 'False'} : Bool;   // Delay Send To VD
      InitSend { ExternalAccessible := 'False'; ExternalVisible := 'False'; ExternalWritable := 'False'} : Bool;   // Init Send
      ResetSendDone { ExternalAccessible := 'False'; ExternalVisible := 'False'; ExternalWritable := 'False'} : Bool;   // Reset Send Done
      ResetAllRequest { ExternalAccessible := 'False'; ExternalVisible := 'False'; ExternalWritable := 'False'} : Bool;   // Reset All Send Requests
      Edge { ExternalAccessible := 'False'; ExternalVisible := 'False'; ExternalWritable := 'False'} : Array[1..64] of Bool;   // Array
      SendDBNbr { ExternalAccessible := 'False'; ExternalVisible := 'False'; ExternalWritable := 'False'} : Int;   // Pointer
      SendDBBufNbr { ExternalAccessible := 'False'; ExternalVisible := 'False'; ExternalWritable := 'False'} : Int;   // Pointer
      AlarmPointer { ExternalAccessible := 'False'; ExternalVisible := 'False'; ExternalWritable := 'False'} : Word;   // Pointer
      AlarmLength { ExternalAccessible := 'False'; ExternalVisible := 'False'; ExternalWritable := 'False'} : Word;   // Pointer
      SendLength { ExternalAccessible := 'False'; ExternalVisible := 'False'; ExternalWritable := 'False'} : Word;   // Pointer
      SendDoneArr { ExternalAccessible := 'False'; ExternalVisible := 'False'; ExternalWritable := 'False'} : Array[0..1] of DWord;   // Array Send Done
   END_VAR
   VAR
      _DelaySend { ExternalAccessible := 'False'; ExternalVisible := 'False'; ExternalWritable := 'False'; S7_SetPoint := 'True'} : "LTimer";   // FB
      _LMDBToDBGen { ExternalAccessible := 'False'; ExternalVisible := 'False'; ExternalWritable := 'False'; S7_SetPoint := 'True'} : "LMDBToDB";   // FB
      _LMDBToDBMZ1 { ExternalAccessible := 'False'; ExternalVisible := 'False'; ExternalWritable := 'False'; S7_SetPoint := 'True'} : "LMDBToDB";   // FB
      _LMDBToDBMZ2 { ExternalAccessible := 'False'; ExternalVisible := 'False'; ExternalWritable := 'False'; S7_SetPoint := 'True'} : "LMDBToDB";   // FB
      _LMDBToDBMZ3 { ExternalAccessible := 'False'; ExternalVisible := 'False'; ExternalWritable := 'False'; S7_SetPoint := 'True'} : "LMDBToDB";   // FB
      _LMDBToDBMZ4 { ExternalAccessible := 'False'; ExternalVisible := 'False'; ExternalWritable := 'False'; S7_SetPoint := 'True'} : "LMDBToDB";   // FB
      _LMDBToDBMZ5 { ExternalAccessible := 'False'; ExternalVisible := 'False'; ExternalWritable := 'False'; S7_SetPoint := 'True'} : "LMDBToDB";   // FB
      _LMDBToDBMZ6 { ExternalAccessible := 'False'; ExternalVisible := 'False'; ExternalWritable := 'False'; S7_SetPoint := 'True'} : "LMDBToDB";   // FB
      _LMDBToDBMZ7 { ExternalAccessible := 'False'; ExternalVisible := 'False'; ExternalWritable := 'False'; S7_SetPoint := 'True'} : "LMDBToDB";   // FB
      _LMDBToDBMZ8 { ExternalAccessible := 'False'; ExternalVisible := 'False'; ExternalWritable := 'False'; S7_SetPoint := 'True'} : "LMDBToDB";   // FB
      _LMDBToDBMZ9 { ExternalAccessible := 'False'; ExternalVisible := 'False'; ExternalWritable := 'False'; S7_SetPoint := 'True'} : "LMDBToDB";   // FB
      _LMDBToDBMZ10 { ExternalAccessible := 'False'; ExternalVisible := 'False'; ExternalWritable := 'False'; S7_SetPoint := 'True'} : "LMDBToDB";   // FB
      _LMDBToDBMZ11 { ExternalAccessible := 'False'; ExternalVisible := 'False'; ExternalWritable := 'False'; S7_SetPoint := 'True'} : "LMDBToDB";   // FB
      _LMDBToDBMZ12 { ExternalAccessible := 'False'; ExternalVisible := 'False'; ExternalWritable := 'False'; S7_SetPoint := 'True'} : "LMDBToDB";   // FB
      _LMDBToDBMZ13 { ExternalAccessible := 'False'; ExternalVisible := 'False'; ExternalWritable := 'False'; S7_SetPoint := 'True'} : "LMDBToDB";   // FB
      _LMDBToDBMZ14 { ExternalAccessible := 'False'; ExternalVisible := 'False'; ExternalWritable := 'False'; S7_SetPoint := 'True'} : "LMDBToDB";   // FB
      _LDBCheckGen { ExternalAccessible := 'False'; ExternalVisible := 'False'; ExternalWritable := 'False'; S7_SetPoint := 'True'} : "LDBCheck";   // FB
      _LDBCheckMZ1 { ExternalAccessible := 'False'; ExternalVisible := 'False'; ExternalWritable := 'False'; S7_SetPoint := 'True'} : "LDBCheck";   // FB
      _LDBCheckMZ2 { ExternalAccessible := 'False'; ExternalVisible := 'False'; ExternalWritable := 'False'; S7_SetPoint := 'True'} : "LDBCheck";   // FB
      _LDBCheckMZ3 { ExternalAccessible := 'False'; ExternalVisible := 'False'; ExternalWritable := 'False'; S7_SetPoint := 'True'} : "LDBCheck";   // FB
      _LDBCheckMZ4 { ExternalAccessible := 'False'; ExternalVisible := 'False'; ExternalWritable := 'False'; S7_SetPoint := 'True'} : "LDBCheck";   // FB
      _LDBCheckMZ5 { ExternalAccessible := 'False'; ExternalVisible := 'False'; ExternalWritable := 'False'; S7_SetPoint := 'True'} : "LDBCheck";   // FB
      _LDBCheckMZ6 { ExternalAccessible := 'False'; ExternalVisible := 'False'; ExternalWritable := 'False'; S7_SetPoint := 'True'} : "LDBCheck";   // FB
      _LDBCheckMZ7 { ExternalAccessible := 'False'; ExternalVisible := 'False'; ExternalWritable := 'False'; S7_SetPoint := 'True'} : "LDBCheck";   // FB
      _LDBCheckMZ8 { ExternalAccessible := 'False'; ExternalVisible := 'False'; ExternalWritable := 'False'; S7_SetPoint := 'True'} : "LDBCheck";   // FB
      _LDBCheckMZ9 { ExternalAccessible := 'False'; ExternalVisible := 'False'; ExternalWritable := 'False'; S7_SetPoint := 'True'} : "LDBCheck";   // FB
      _LDBCheckMZ10 { ExternalAccessible := 'False'; ExternalVisible := 'False'; ExternalWritable := 'False'; S7_SetPoint := 'True'} : "LDBCheck";   // FB
      _LDBCheckMZ11 { ExternalAccessible := 'False'; ExternalVisible := 'False'; ExternalWritable := 'False'; S7_SetPoint := 'True'} : "LDBCheck";   // FB
      _LDBCheckMZ12 { ExternalAccessible := 'False'; ExternalVisible := 'False'; ExternalWritable := 'False'; S7_SetPoint := 'True'} : "LDBCheck";   // FB
      _LDBCheckMZ13 { ExternalAccessible := 'False'; ExternalVisible := 'False'; ExternalWritable := 'False'; S7_SetPoint := 'True'} : "LDBCheck";   // FB
      _LDBCheckMZ14 { ExternalAccessible := 'False'; ExternalVisible := 'False'; ExternalWritable := 'False'; S7_SetPoint := 'True'} : "LDBCheck";   // FB
   END_VAR
   VAR DB_SPECIFIC
      _SendDoneReset { ExternalAccessible := 'False'; ExternalVisible := 'False'; ExternalWritable := 'False'; S7_SetPoint := 'True'} : TON_TIME;   // FB
      Filter { ExternalAccessible := 'False'; ExternalVisible := 'False'; ExternalWritable := 'False'} : Array[1..16] of Bool;   // Array
      _FilterGen { ExternalAccessible := 'False'; ExternalVisible := 'False'; ExternalWritable := 'False'; S7_SetPoint := 'True'} : TON_TIME;   // FB
      _FilterMZ1 { ExternalAccessible := 'False'; ExternalVisible := 'False'; ExternalWritable := 'False'; S7_SetPoint := 'True'} : TON_TIME;   // FB
      _FilterMZ2 { ExternalAccessible := 'False'; ExternalVisible := 'False'; ExternalWritable := 'False'; S7_SetPoint := 'True'} : TON_TIME;   // FB
      _FilterMZ3 { ExternalAccessible := 'False'; ExternalVisible := 'False'; ExternalWritable := 'False'; S7_SetPoint := 'True'} : TON_TIME;   // FB
      _FilterMZ4 { ExternalAccessible := 'False'; ExternalVisible := 'False'; ExternalWritable := 'False'; S7_SetPoint := 'True'} : TON_TIME;   // FB
      _FilterMZ5 { ExternalAccessible := 'False'; ExternalVisible := 'False'; ExternalWritable := 'False'; S7_SetPoint := 'True'} : TON_TIME;   // FB
      _FilterMZ6 { ExternalAccessible := 'False'; ExternalVisible := 'False'; ExternalWritable := 'False'; S7_SetPoint := 'True'} : TON_TIME;   // FB
      _FilterMZ7 { ExternalAccessible := 'False'; ExternalVisible := 'False'; ExternalWritable := 'False'; S7_SetPoint := 'True'} : TON_TIME;   // FB
      _FilterMZ8 { ExternalAccessible := 'False'; ExternalVisible := 'False'; ExternalWritable := 'False'; S7_SetPoint := 'True'} : TON_TIME;   // FB
      _FilterMZ9 { ExternalAccessible := 'False'; ExternalVisible := 'False'; ExternalWritable := 'False'; S7_SetPoint := 'True'} : TON_TIME;   // FB
      _FilterMZ10 { ExternalAccessible := 'False'; ExternalVisible := 'False'; ExternalWritable := 'False'; S7_SetPoint := 'True'} : TON_TIME;   // FB
      _FilterMZ11 { ExternalAccessible := 'False'; ExternalVisible := 'False'; ExternalWritable := 'False'; S7_SetPoint := 'True'} : TON_TIME;   // FB
      _FilterMZ12 { ExternalAccessible := 'False'; ExternalVisible := 'False'; ExternalWritable := 'False'; S7_SetPoint := 'True'} : TON_TIME;   // FB
      _FilterMZ13 { ExternalAccessible := 'False'; ExternalVisible := 'False'; ExternalWritable := 'False'; S7_SetPoint := 'True'} : TON_TIME;   // FB
      _FilterMZ14 { ExternalAccessible := 'False'; ExternalVisible := 'False'; ExternalWritable := 'False'; S7_SetPoint := 'True'} : TON_TIME;   // FB
      _InitSend { ExternalAccessible := 'False'; ExternalVisible := 'False'; ExternalWritable := 'False'; S7_SetPoint := 'True'} : TON_TIME;   // FB
      GenDBLenghtOk { ExternalAccessible := 'False'; ExternalVisible := 'False'; ExternalWritable := 'False'} : Bool;   // DB Length Ok
      MZ1DBLenghtOk { ExternalAccessible := 'False'; ExternalVisible := 'False'; ExternalWritable := 'False'} : Bool;   // DB Length Ok
      MZ2DBLenghtOk { ExternalAccessible := 'False'; ExternalVisible := 'False'; ExternalWritable := 'False'} : Bool;   // DB Length Ok
      MZ3DBLenghtOk { ExternalAccessible := 'False'; ExternalVisible := 'False'; ExternalWritable := 'False'} : Bool;   // DB Length Ok
      MZ4DBLenghtOk { ExternalAccessible := 'False'; ExternalVisible := 'False'; ExternalWritable := 'False'} : Bool;   // DB Length Ok
      MZ5DBLenghtOk { ExternalAccessible := 'False'; ExternalVisible := 'False'; ExternalWritable := 'False'} : Bool;   // DB Length Ok
      MZ6DBLenghtOk { ExternalAccessible := 'False'; ExternalVisible := 'False'; ExternalWritable := 'False'} : Bool;   // DB Length Ok
      MZ7DBLenghtOk { ExternalAccessible := 'False'; ExternalVisible := 'False'; ExternalWritable := 'False'} : Bool;   // DB Length Ok
      MZ8DBLenghtOk { ExternalAccessible := 'False'; ExternalVisible := 'False'; ExternalWritable := 'False'} : Bool;   // DB Length Ok
      MZ9DBLenghtOk { ExternalAccessible := 'False'; ExternalVisible := 'False'; ExternalWritable := 'False'} : Bool;   // DB Length Ok
      MZ10DBLenghtOk { ExternalAccessible := 'False'; ExternalVisible := 'False'; ExternalWritable := 'False'} : Bool;   // DB Length Ok
      MZ11DBLenghtOk { ExternalAccessible := 'False'; ExternalVisible := 'False'; ExternalWritable := 'False'} : Bool;   // DB Length Ok
      MZ12DBLenghtOk { ExternalAccessible := 'False'; ExternalVisible := 'False'; ExternalWritable := 'False'} : Bool;   // DB Length Ok
      MZ13DBLenghtOk { ExternalAccessible := 'False'; ExternalVisible := 'False'; ExternalWritable := 'False'} : Bool;   // DB Length Ok
      MZ14DBLenghtOk { ExternalAccessible := 'False'; ExternalVisible := 'False'; ExternalWritable := 'False'} : Bool;   // DB Length Ok
      MZ15DBLenghtOk { ExternalAccessible := 'False'; ExternalVisible := 'False'; ExternalWritable := 'False'} : Bool;   // DB Length Ok
      MZ16DBLenghtOk { ExternalAccessible := 'False'; ExternalVisible := 'False'; ExternalWritable := 'False'} : Bool;   // DB Length Ok
      GenDBLength { ExternalAccessible := 'False'; ExternalVisible := 'False'; ExternalWritable := 'False'} : Word;   // DB Header
      GenDBNumber { ExternalAccessible := 'False'; ExternalVisible := 'False'; ExternalWritable := 'False'} : Word;   // DB Header
      MZ1DBLength { ExternalAccessible := 'False'; ExternalVisible := 'False'; ExternalWritable := 'False'} : Word;   // DB Header
      MZ1DBNumber { ExternalAccessible := 'False'; ExternalVisible := 'False'; ExternalWritable := 'False'} : Word;   // DB Header
      MZ2DBLength { ExternalAccessible := 'False'; ExternalVisible := 'False'; ExternalWritable := 'False'} : Word;   // DB Header
      MZ2DBNumber { ExternalAccessible := 'False'; ExternalVisible := 'False'; ExternalWritable := 'False'} : Word;   // DB Header
      MZ3DBLength { ExternalAccessible := 'False'; ExternalVisible := 'False'; ExternalWritable := 'False'} : Word;   // DB Header
      MZ3DBNumber { ExternalAccessible := 'False'; ExternalVisible := 'False'; ExternalWritable := 'False'} : Word;   // DB Header
      MZ4DBLength { ExternalAccessible := 'False'; ExternalVisible := 'False'; ExternalWritable := 'False'} : Word;   // DB Header
      MZ4DBNumber { ExternalAccessible := 'False'; ExternalVisible := 'False'; ExternalWritable := 'False'} : Word;   // DB Header
      MZ5DBLength { ExternalAccessible := 'False'; ExternalVisible := 'False'; ExternalWritable := 'False'} : Word;   // DB Header
      MZ5DBNumber { ExternalAccessible := 'False'; ExternalVisible := 'False'; ExternalWritable := 'False'} : Word;   // DB Header
      MZ6DBLength { ExternalAccessible := 'False'; ExternalVisible := 'False'; ExternalWritable := 'False'} : Word;   // DB Header
      MZ6DBNumber { ExternalAccessible := 'False'; ExternalVisible := 'False'; ExternalWritable := 'False'} : Word;   // DB Header
      MZ7DBLength { ExternalAccessible := 'False'; ExternalVisible := 'False'; ExternalWritable := 'False'} : Word;   // DB Header
      MZ7DBNumber { ExternalAccessible := 'False'; ExternalVisible := 'False'; ExternalWritable := 'False'} : Word;   // DB Header
      MZ8DBLength { ExternalAccessible := 'False'; ExternalVisible := 'False'; ExternalWritable := 'False'} : Word;   // DB Header
      MZ8DBNumber { ExternalAccessible := 'False'; ExternalVisible := 'False'; ExternalWritable := 'False'} : Word;   // DB Header
      MZ9DBLength { ExternalAccessible := 'False'; ExternalVisible := 'False'; ExternalWritable := 'False'} : Word;   // DB Header
      MZ9DBNumber { ExternalAccessible := 'False'; ExternalVisible := 'False'; ExternalWritable := 'False'} : Word;   // DB Header
      MZ10DBLength { ExternalAccessible := 'False'; ExternalVisible := 'False'; ExternalWritable := 'False'} : Word;   // DB Header
      MZ10DBNumber { ExternalAccessible := 'False'; ExternalVisible := 'False'; ExternalWritable := 'False'} : Word;   // DB Header
      MZ11DBLength { ExternalAccessible := 'False'; ExternalVisible := 'False'; ExternalWritable := 'False'} : Word;   // DB Header
      MZ11DBNumber { ExternalAccessible := 'False'; ExternalVisible := 'False'; ExternalWritable := 'False'} : Word;   // DB Header
      MZ12DBLength { ExternalAccessible := 'False'; ExternalVisible := 'False'; ExternalWritable := 'False'} : Word;   // DB Header
      MZ12DBNumber { ExternalAccessible := 'False'; ExternalVisible := 'False'; ExternalWritable := 'False'} : Word;   // DB Header
      MZ13DBLength { ExternalAccessible := 'False'; ExternalVisible := 'False'; ExternalWritable := 'False'} : Word;   // DB Header
      MZ13DBNumber { ExternalAccessible := 'False'; ExternalVisible := 'False'; ExternalWritable := 'False'} : Word;   // DB Header
      MZ14DBLength { ExternalAccessible := 'False'; ExternalVisible := 'False'; ExternalWritable := 'False'} : Word;   // DB Header
      MZ14DBNumber { ExternalAccessible := 'False'; ExternalVisible := 'False'; ExternalWritable := 'False'} : Word;   // DB Header
      PLCAlarms { ExternalAccessible := 'False'; ExternalVisible := 'False'; ExternalWritable := 'False'; S7_SetPoint := 'True'} : "PLCAlarms";   // Alarm Handling
   END_VAR
   VAR_TEMP
      BPtr : Any;   // Temp
      SPtr : Any;   // Temp
      Pointer : Word;   // Temp
      F : Word;
      GenDBLenghtCompare : Word;   // Temp
      MZ1DBLenghtCompare : Word;   // Temp
      MZ2DBLenghtCompare : Word;   // Temp
      MZ3DBLenghtCompare : Word;   // Temp
      MZ4DBLenghtCompare : Word;   // Temp
      MZ5DBLenghtCompare : Word;   // Temp
      MZ6DBLenghtCompare : Word;   // Temp
      MZ7DBLenghtCompare : Word;   // Temp
      MZ8DBLenghtCompare : Word;   // Temp
      MZ9DBLenghtCompare : Word;   // Temp
      MZ10DBLenghtCompare : Word;   // Temp
      MZ11DBLenghtCompare : Word;   // Temp
      MZ12DBLenghtCompare : Word;   // Temp
      MZ13DBLenghtCompare : Word;   // Temp
      MZ14DBLenghtCompare : Word;   // Temp
      GenOk : Bool;   // Temp
      MZ1Ok : Bool;   // Temp
      MZ2Ok : Bool;   // Temp
      MZ3Ok : Bool;   // Temp
      MZ4Ok : Bool;   // Temp
      MZ5Ok : Bool;   // Temp
      MZ6Ok : Bool;   // Temp
      MZ7Ok : Bool;   // Temp
      MZ8Ok : Bool;   // Temp
      MZ9Ok : Bool;   // Temp
      MZ10Ok : Bool;   // Temp
      MZ11Ok : Bool;   // Temp
      MZ12Ok : Bool;   // Temp
      MZ13Ok : Bool;   // Temp
      MZ14Ok : Bool;   // Temp
   END_VAR
   VAR_TEMP   // added for the SCL form of the ladder/FBD networks
      _w1 : Bool;
   END_VAR
BEGIN

REGION Network 1: **** 3.1 - Communication - Other Systems **** Request Event To VD
   // Request Send To VD
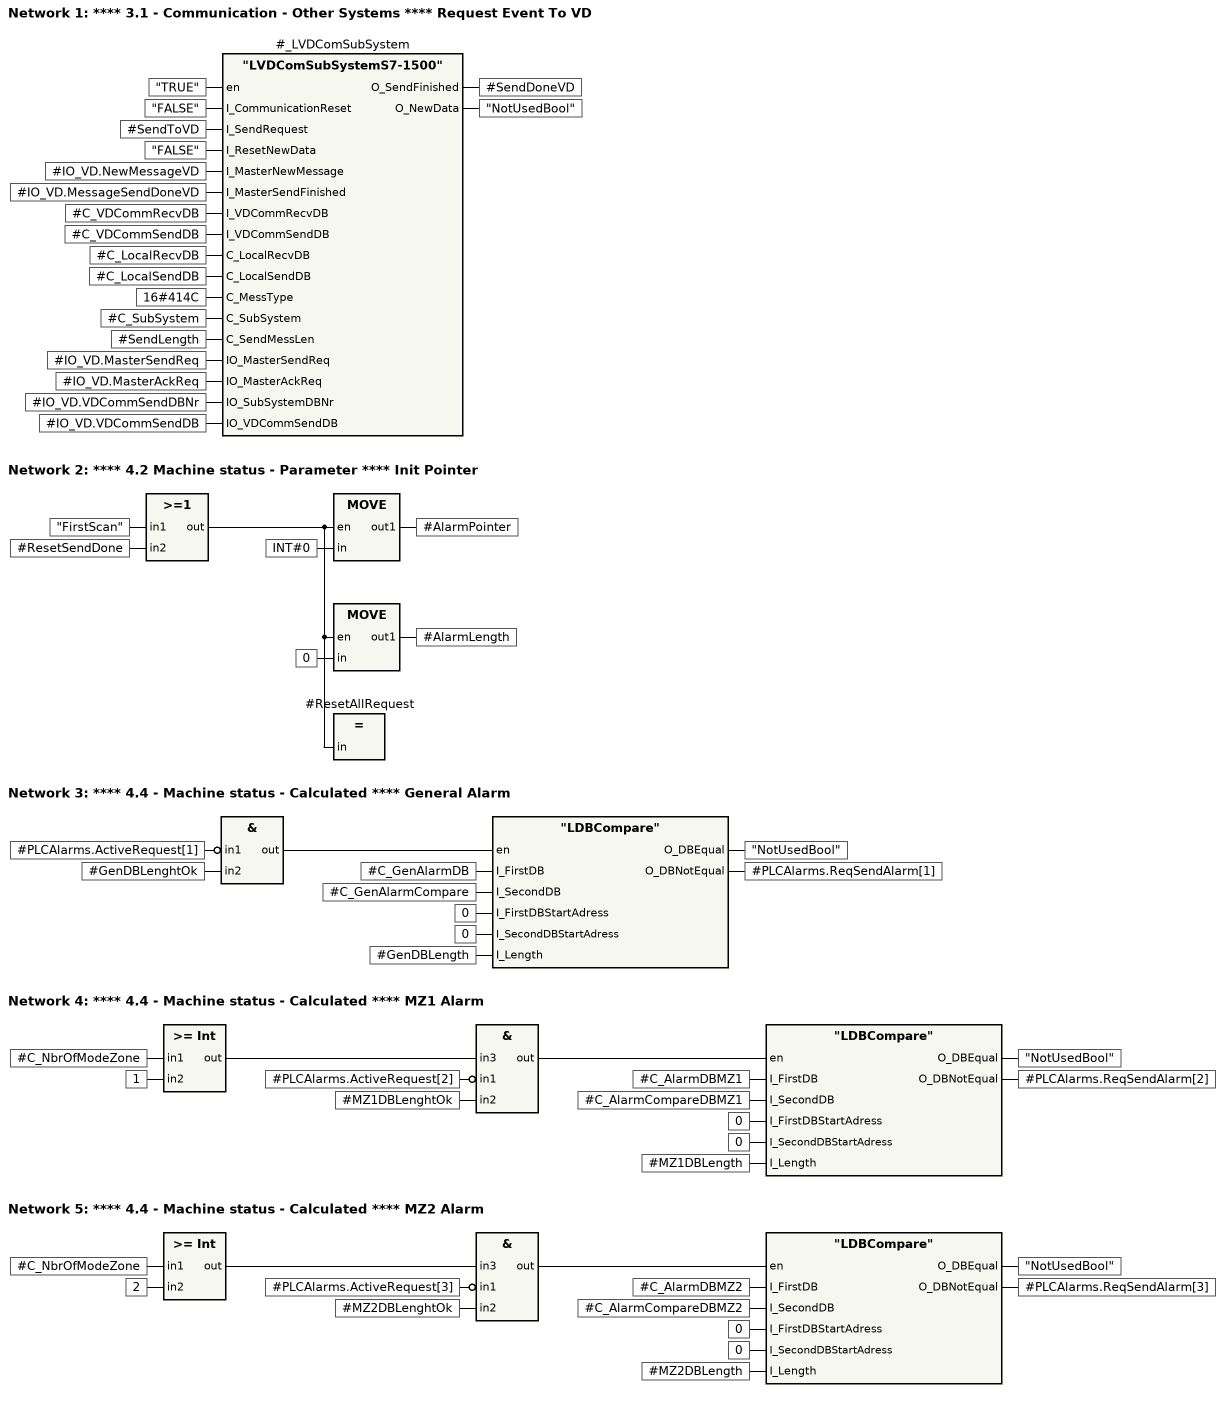
   IF "TRUE" THEN
       #_LVDComSubSystem(I_CommunicationReset := "FALSE",   // "LVDComSubSystemS7-1500"
                         I_SendRequest := #SendToVD,
                         I_ResetNewData := "FALSE",
                         I_MasterNewMessage := #IO_VD.NewMessageVD,
                         I_MasterSendFinished := #IO_VD.MessageSendDoneVD,
                         I_VDCommRecvDB := #C_VDCommRecvDB,
                         I_VDCommSendDB := #C_VDCommSendDB,
                         C_LocalRecvDB := #C_LocalRecvDB,
                         C_LocalSendDB := #C_LocalSendDB,
                         C_MessType := 16#414C,
                         C_SubSystem := #C_SubSystem,
                         C_SendMessLen := #SendLength,
                         IO_MasterSendReq := #IO_VD.MasterSendReq,
                         IO_MasterAckReq := #IO_VD.MasterAckReq,
                         IO_SubSystemDBNr := #IO_VD.VDCommSendDBNr,
                         IO_VDCommSendDB := #IO_VD.VDCommSendDB,
                         O_SendFinished => #SendDoneVD,
                         O_NewData => "NotUsedBool");
   END_IF;
END_REGION

REGION Network 2: **** 4.2 Machine status - Parameter **** Init Pointer
   // Init Pointer
   #_w1 := "FirstScan" OR #ResetSendDone;
   IF #_w1 THEN
       #AlarmPointer := INT#0;
       #AlarmLength := 0;
   END_IF;
   #ResetAllRequest := #_w1;
END_REGION

REGION Network 3: **** 4.4 - Machine status - Calculated **** General Alarm
   // Check If There Is New Alarms
   IF NOT #PLCAlarms.ActiveRequest[1] AND #GenDBLenghtOk THEN
       "LDBCompare"(I_FirstDB := #C_GenAlarmDB,
                    I_SecondDB := #C_GenAlarmCompare,
                    I_FirstDBStartAdress := 0,
                    I_SecondDBStartAdress := 0,
                    I_Length := #GenDBLength,
                    O_DBEqual => "NotUsedBool",
                    O_DBNotEqual => #PLCAlarms.ReqSendAlarm[1]);
   END_IF;
END_REGION

REGION Network 4: **** 4.4 - Machine status - Calculated **** MZ1 Alarm
   // Check If There Is New Alarms
   IF (#C_NbrOfModeZone >= 1) AND NOT #PLCAlarms.ActiveRequest[2] AND #MZ1DBLenghtOk THEN
       "LDBCompare"(I_FirstDB := #C_AlarmDBMZ1,
                    I_SecondDB := #C_AlarmCompareDBMZ1,
                    I_FirstDBStartAdress := 0,
                    I_SecondDBStartAdress := 0,
                    I_Length := #MZ1DBLength,
                    O_DBEqual => "NotUsedBool",
                    O_DBNotEqual => #PLCAlarms.ReqSendAlarm[2]);
   END_IF;
END_REGION

REGION Network 5: **** 4.4 - Machine status - Calculated **** MZ2 Alarm
   // Check If There Is New Alarms
   IF (#C_NbrOfModeZone >= 2) AND NOT #PLCAlarms.ActiveRequest[3] AND #MZ2DBLenghtOk THEN
       "LDBCompare"(I_FirstDB := #C_AlarmDBMZ2,
                    I_SecondDB := #C_AlarmCompareDBMZ2,
                    I_FirstDBStartAdress := 0,
                    I_SecondDBStartAdress := 0,
                    I_Length := #MZ2DBLength,
                    O_DBEqual => "NotUsedBool",
                    O_DBNotEqual => #PLCAlarms.ReqSendAlarm[3]);
   END_IF;
END_REGION

REGION Network 6: **** 4.4 - Machine status - Calculated **** MZ3 Alarm
   // Check If There Is New Alarms
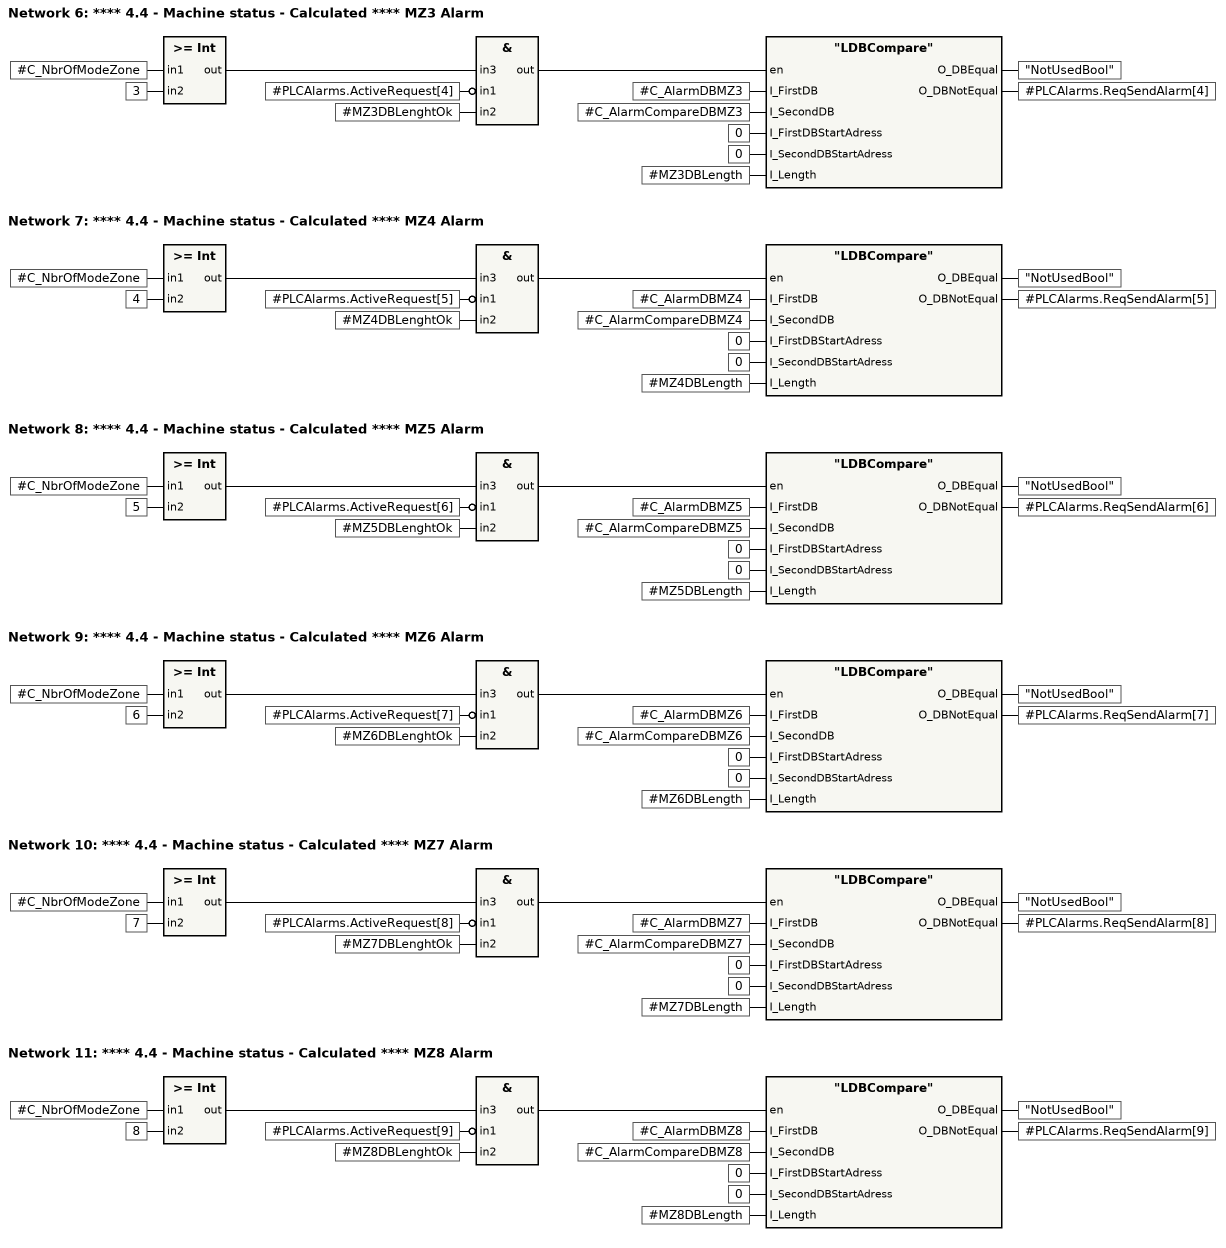
   IF (#C_NbrOfModeZone >= 3) AND NOT #PLCAlarms.ActiveRequest[4] AND #MZ3DBLenghtOk THEN
       "LDBCompare"(I_FirstDB := #C_AlarmDBMZ3,
                    I_SecondDB := #C_AlarmCompareDBMZ3,
                    I_FirstDBStartAdress := 0,
                    I_SecondDBStartAdress := 0,
                    I_Length := #MZ3DBLength,
                    O_DBEqual => "NotUsedBool",
                    O_DBNotEqual => #PLCAlarms.ReqSendAlarm[4]);
   END_IF;
END_REGION

REGION Network 7: **** 4.4 - Machine status - Calculated **** MZ4 Alarm
   // Check If There Is New Alarms
   IF (#C_NbrOfModeZone >= 4) AND NOT #PLCAlarms.ActiveRequest[5] AND #MZ4DBLenghtOk THEN
       "LDBCompare"(I_FirstDB := #C_AlarmDBMZ4,
                    I_SecondDB := #C_AlarmCompareDBMZ4,
                    I_FirstDBStartAdress := 0,
                    I_SecondDBStartAdress := 0,
                    I_Length := #MZ4DBLength,
                    O_DBEqual => "NotUsedBool",
                    O_DBNotEqual => #PLCAlarms.ReqSendAlarm[5]);
   END_IF;
END_REGION

REGION Network 8: **** 4.4 - Machine status - Calculated **** MZ5 Alarm
   // Check If There Is New Alarms
   IF (#C_NbrOfModeZone >= 5) AND NOT #PLCAlarms.ActiveRequest[6] AND #MZ5DBLenghtOk THEN
       "LDBCompare"(I_FirstDB := #C_AlarmDBMZ5,
                    I_SecondDB := #C_AlarmCompareDBMZ5,
                    I_FirstDBStartAdress := 0,
                    I_SecondDBStartAdress := 0,
                    I_Length := #MZ5DBLength,
                    O_DBEqual => "NotUsedBool",
                    O_DBNotEqual => #PLCAlarms.ReqSendAlarm[6]);
   END_IF;
END_REGION

REGION Network 9: **** 4.4 - Machine status - Calculated **** MZ6 Alarm
   // Check If There Is New Alarms
   IF (#C_NbrOfModeZone >= 6) AND NOT #PLCAlarms.ActiveRequest[7] AND #MZ6DBLenghtOk THEN
       "LDBCompare"(I_FirstDB := #C_AlarmDBMZ6,
                    I_SecondDB := #C_AlarmCompareDBMZ6,
                    I_FirstDBStartAdress := 0,
                    I_SecondDBStartAdress := 0,
                    I_Length := #MZ6DBLength,
                    O_DBEqual => "NotUsedBool",
                    O_DBNotEqual => #PLCAlarms.ReqSendAlarm[7]);
   END_IF;
END_REGION

REGION Network 10: **** 4.4 - Machine status - Calculated **** MZ7 Alarm
   // Check If There Is New Alarms
   IF (#C_NbrOfModeZone >= 7) AND NOT #PLCAlarms.ActiveRequest[8] AND #MZ7DBLenghtOk THEN
       "LDBCompare"(I_FirstDB := #C_AlarmDBMZ7,
                    I_SecondDB := #C_AlarmCompareDBMZ7,
                    I_FirstDBStartAdress := 0,
                    I_SecondDBStartAdress := 0,
                    I_Length := #MZ7DBLength,
                    O_DBEqual => "NotUsedBool",
                    O_DBNotEqual => #PLCAlarms.ReqSendAlarm[8]);
   END_IF;
END_REGION

REGION Network 11: **** 4.4 - Machine status - Calculated **** MZ8 Alarm
   // Check If There Is New Alarms
   IF (#C_NbrOfModeZone >= 8) AND NOT #PLCAlarms.ActiveRequest[9] AND #MZ8DBLenghtOk THEN
       "LDBCompare"(I_FirstDB := #C_AlarmDBMZ8,
                    I_SecondDB := #C_AlarmCompareDBMZ8,
                    I_FirstDBStartAdress := 0,
                    I_SecondDBStartAdress := 0,
                    I_Length := #MZ8DBLength,
                    O_DBEqual => "NotUsedBool",
                    O_DBNotEqual => #PLCAlarms.ReqSendAlarm[9]);
   END_IF;
END_REGION

REGION Network 12: **** 4.4 - Machine status - Calculated **** MZ9 Alarm
   // Check If There Is New Alarms
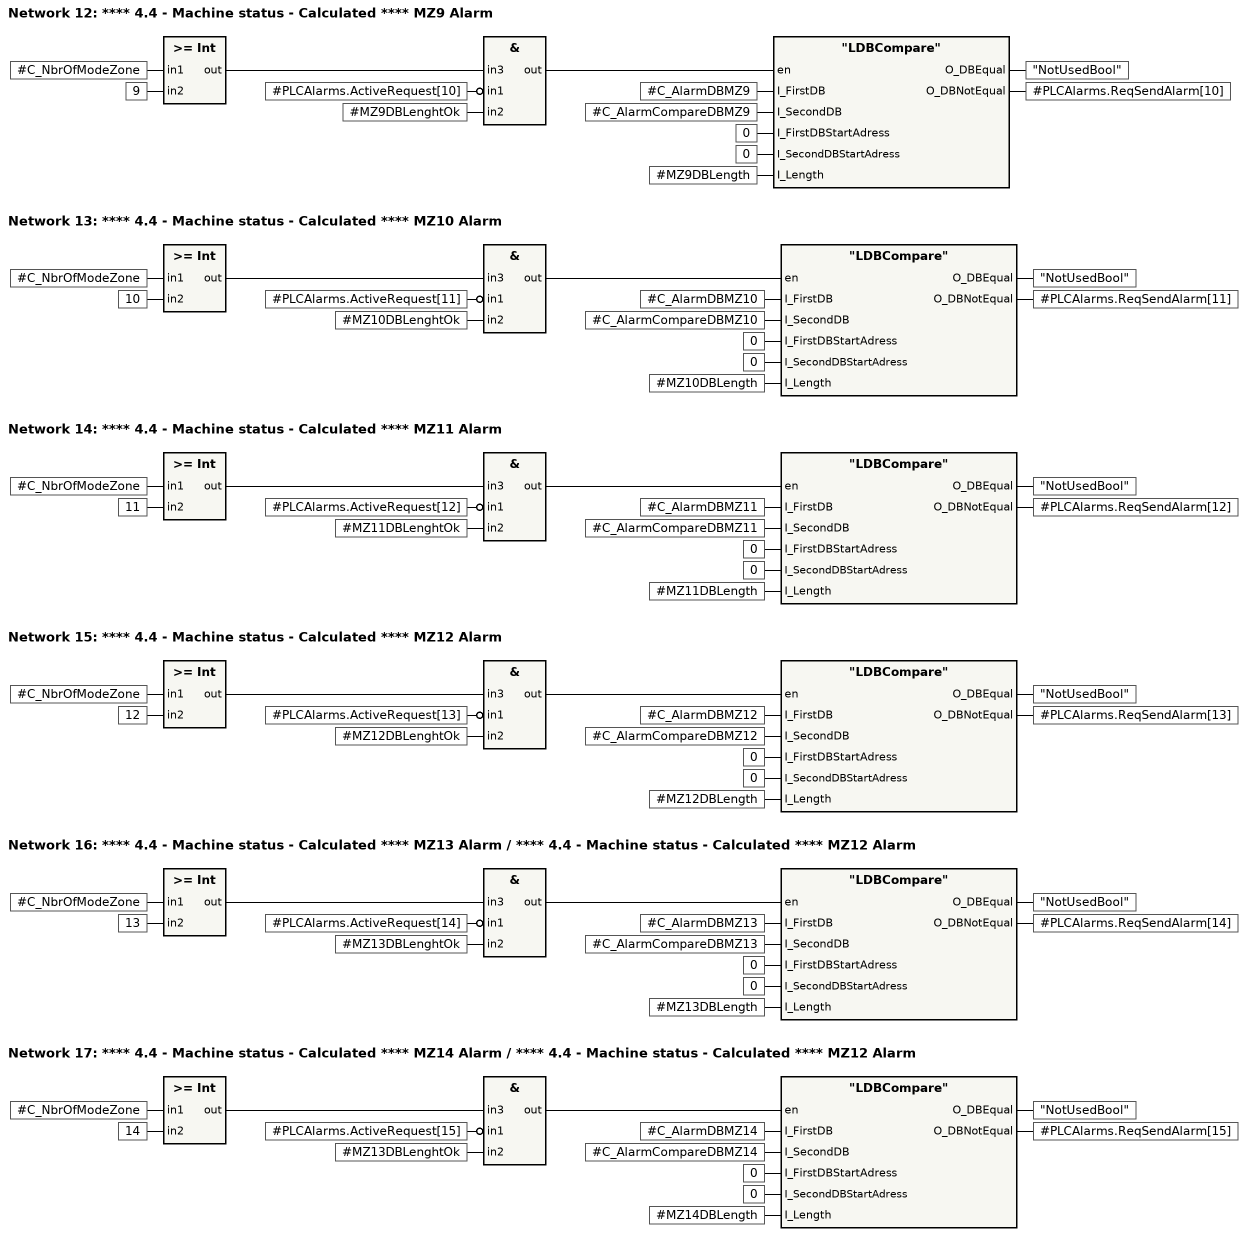
   IF (#C_NbrOfModeZone >= 9) AND NOT #PLCAlarms.ActiveRequest[10] AND #MZ9DBLenghtOk THEN
       "LDBCompare"(I_FirstDB := #C_AlarmDBMZ9,
                    I_SecondDB := #C_AlarmCompareDBMZ9,
                    I_FirstDBStartAdress := 0,
                    I_SecondDBStartAdress := 0,
                    I_Length := #MZ9DBLength,
                    O_DBEqual => "NotUsedBool",
                    O_DBNotEqual => #PLCAlarms.ReqSendAlarm[10]);
   END_IF;
END_REGION

REGION Network 13: **** 4.4 - Machine status - Calculated **** MZ10 Alarm
   // Check If There Is New Alarms
   IF (#C_NbrOfModeZone >= 10) AND NOT #PLCAlarms.ActiveRequest[11] AND #MZ10DBLenghtOk THEN
       "LDBCompare"(I_FirstDB := #C_AlarmDBMZ10,
                    I_SecondDB := #C_AlarmCompareDBMZ10,
                    I_FirstDBStartAdress := 0,
                    I_SecondDBStartAdress := 0,
                    I_Length := #MZ10DBLength,
                    O_DBEqual => "NotUsedBool",
                    O_DBNotEqual => #PLCAlarms.ReqSendAlarm[11]);
   END_IF;
END_REGION

REGION Network 14: **** 4.4 - Machine status - Calculated **** MZ11 Alarm
   // Check If There Is New Alarms
   IF (#C_NbrOfModeZone >= 11) AND NOT #PLCAlarms.ActiveRequest[12] AND #MZ11DBLenghtOk THEN
       "LDBCompare"(I_FirstDB := #C_AlarmDBMZ11,
                    I_SecondDB := #C_AlarmCompareDBMZ11,
                    I_FirstDBStartAdress := 0,
                    I_SecondDBStartAdress := 0,
                    I_Length := #MZ11DBLength,
                    O_DBEqual => "NotUsedBool",
                    O_DBNotEqual => #PLCAlarms.ReqSendAlarm[12]);
   END_IF;
END_REGION

REGION Network 15: **** 4.4 - Machine status - Calculated **** MZ12 Alarm
   // Check If There Is New Alarms
   IF (#C_NbrOfModeZone >= 12) AND NOT #PLCAlarms.ActiveRequest[13] AND #MZ12DBLenghtOk THEN
       "LDBCompare"(I_FirstDB := #C_AlarmDBMZ12,
                    I_SecondDB := #C_AlarmCompareDBMZ12,
                    I_FirstDBStartAdress := 0,
                    I_SecondDBStartAdress := 0,
                    I_Length := #MZ12DBLength,
                    O_DBEqual => "NotUsedBool",
                    O_DBNotEqual => #PLCAlarms.ReqSendAlarm[13]);
   END_IF;
END_REGION

REGION Network 16: **** 4.4 - Machine status - Calculated **** MZ13 Alarm / **** 4.4 - Machine status - Calculated **** MZ12 Alarm
   // Check If There Is New Alarms
   IF (#C_NbrOfModeZone >= 13) AND NOT #PLCAlarms.ActiveRequest[14] AND #MZ13DBLenghtOk THEN
       "LDBCompare"(I_FirstDB := #C_AlarmDBMZ13,
                    I_SecondDB := #C_AlarmCompareDBMZ13,
                    I_FirstDBStartAdress := 0,
                    I_SecondDBStartAdress := 0,
                    I_Length := #MZ13DBLength,
                    O_DBEqual => "NotUsedBool",
                    O_DBNotEqual => #PLCAlarms.ReqSendAlarm[14]);
   END_IF;
END_REGION

REGION Network 17: **** 4.4 - Machine status - Calculated **** MZ14 Alarm / **** 4.4 - Machine status - Calculated **** MZ12 Alarm
   // Check If There Is New Alarms
   IF (#C_NbrOfModeZone >= 14) AND NOT #PLCAlarms.ActiveRequest[15] AND #MZ13DBLenghtOk THEN
       "LDBCompare"(I_FirstDB := #C_AlarmDBMZ14,
                    I_SecondDB := #C_AlarmCompareDBMZ14,
                    I_FirstDBStartAdress := 0,
                    I_SecondDBStartAdress := 0,
                    I_Length := #MZ14DBLength,
                    O_DBEqual => "NotUsedBool",
                    O_DBNotEqual => #PLCAlarms.ReqSendAlarm[15]);
   END_IF;
END_REGION

REGION Network 18: **** 4.4 - Machine status - Calculated **** Erase All Requests
   // Erase All Requests
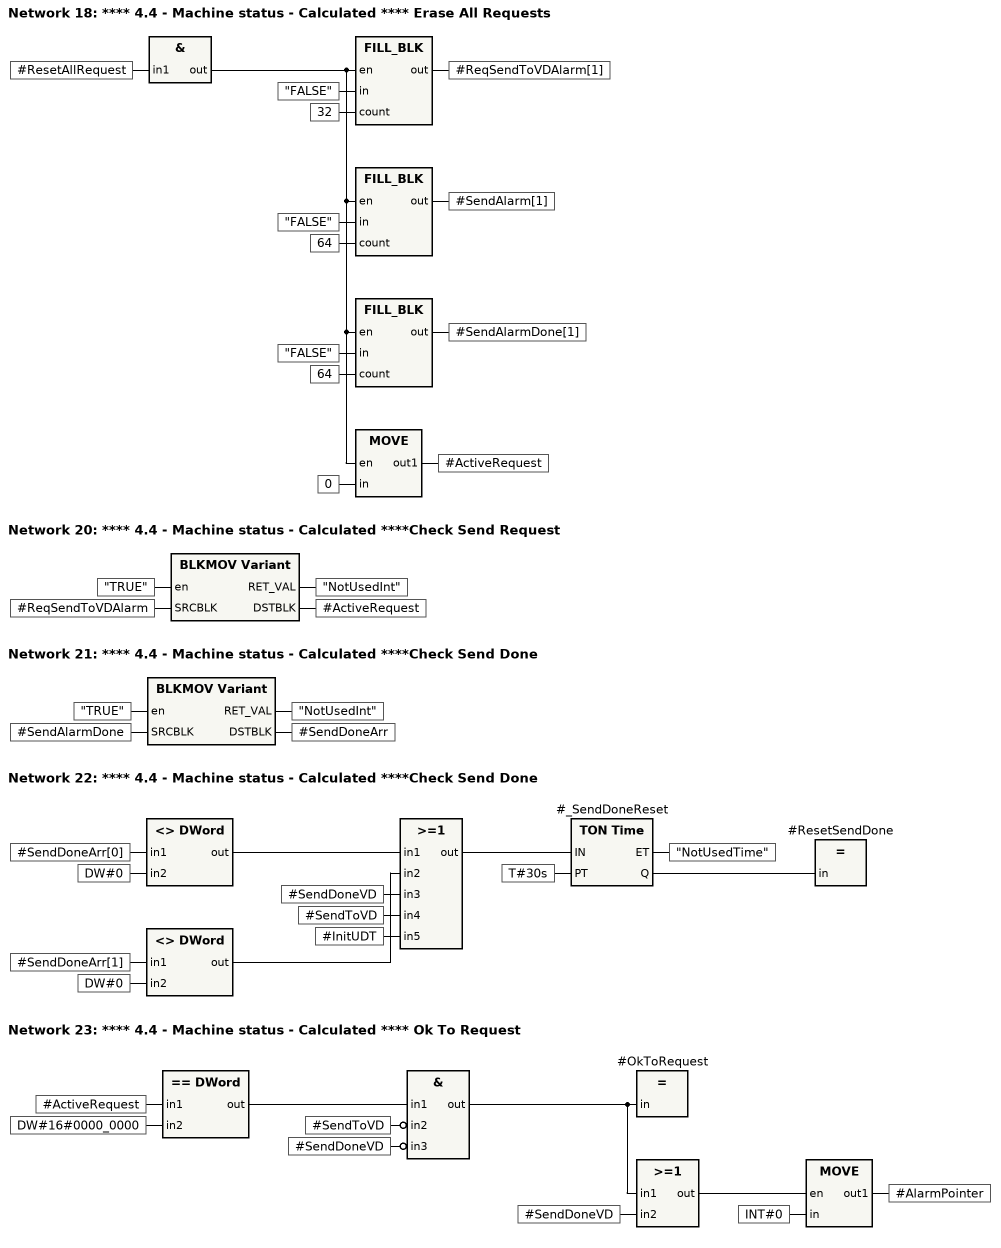
   IF #ResetAllRequest THEN
       FILL_BLK(IN := "FALSE", COUNT := 32, OUT => #ReqSendToVDAlarm[1]);
       FILL_BLK(IN := "FALSE", COUNT := 64, OUT => #SendAlarm[1]);
       FILL_BLK(IN := "FALSE", COUNT := 64, OUT => #SendAlarmDone[1]);
       #ActiveRequest := 0;
   END_IF;
END_REGION

NETWORK
TITLE = **** 4.4 - Machine status - Calculated **** Init UDT
// Init UDT
      A     #ResetAllRequest;
      O     #ResetSendDone;
      JCN   NoInit;
      R     #PLCAlarms.ReqSendAlarm[1];
      R     #PLCAlarms.ReqSendAlarm[2];
      R     #PLCAlarms.ReqSendAlarm[3];
      R     #PLCAlarms.ReqSendAlarm[4];
      R     #PLCAlarms.ReqSendAlarm[5];
      R     #PLCAlarms.ReqSendAlarm[6];
      R     #PLCAlarms.ReqSendAlarm[7];
      R     #PLCAlarms.ReqSendAlarm[8];
      R     #PLCAlarms.ReqSendAlarm[9];
      R     #PLCAlarms.ReqSendAlarm[10];
      R     #PLCAlarms.ReqSendAlarm[11];
      R     #PLCAlarms.ReqSendAlarm[12];
      R     #PLCAlarms.ReqSendAlarm[13];
      R     #PLCAlarms.ReqSendAlarm[14];
      R     #PLCAlarms.ReqSendAlarm[15];
      R     #PLCAlarms.ReqSendAlarm[16];
      R     #PLCAlarms.ReqSendAlarm[17];
      R     #PLCAlarms.ReqSendAlarm[18];
      R     #PLCAlarms.ReqSendAlarm[19];
      R     #PLCAlarms.ReqSendAlarm[20];
      R     #PLCAlarms.ReqSendAlarm[21];
      R     #PLCAlarms.ReqSendAlarm[22];
      R     #PLCAlarms.ReqSendAlarm[23];
      R     #PLCAlarms.ReqSendAlarm[24];
      R     #PLCAlarms.ReqSendAlarm[25];
      R     #PLCAlarms.ReqSendAlarm[26];
      R     #PLCAlarms.ReqSendAlarm[27];
      R     #PLCAlarms.ReqSendAlarm[28];
      R     #PLCAlarms.ReqSendAlarm[29];
      R     #PLCAlarms.ReqSendAlarm[30];
      R     #PLCAlarms.ReqSendAlarm[31];
      R     #PLCAlarms.ReqSendAlarm[32];
      R     #PLCAlarms.ActiveRequest[1];
      R     #PLCAlarms.ActiveRequest[2];
      R     #PLCAlarms.ActiveRequest[3];
      R     #PLCAlarms.ActiveRequest[4];
      R     #PLCAlarms.ActiveRequest[5];
      R     #PLCAlarms.ActiveRequest[6];
      R     #PLCAlarms.ActiveRequest[7];
      R     #PLCAlarms.ActiveRequest[8];
      R     #PLCAlarms.ActiveRequest[9];
      R     #PLCAlarms.ActiveRequest[10];
      R     #PLCAlarms.ActiveRequest[11];
      R     #PLCAlarms.ActiveRequest[12];
      R     #PLCAlarms.ActiveRequest[13];
      R     #PLCAlarms.ActiveRequest[14];
      R     #PLCAlarms.ActiveRequest[15];
      R     #PLCAlarms.ActiveRequest[16];
      R     #PLCAlarms.ActiveRequest[17];
      R     #PLCAlarms.ActiveRequest[18];
      R     #PLCAlarms.ActiveRequest[19];
      R     #PLCAlarms.ActiveRequest[20];
      R     #PLCAlarms.ActiveRequest[21];
      R     #PLCAlarms.ActiveRequest[22];
      R     #PLCAlarms.ActiveRequest[23];
      R     #PLCAlarms.ActiveRequest[24];
      R     #PLCAlarms.ActiveRequest[25];
      R     #PLCAlarms.ActiveRequest[26];
      R     #PLCAlarms.ActiveRequest[27];
      R     #PLCAlarms.ActiveRequest[28];
      R     #PLCAlarms.ActiveRequest[29];
      R     #PLCAlarms.ActiveRequest[30];
      R     #PLCAlarms.ActiveRequest[31];
      R     #PLCAlarms.ActiveRequest[32];

NoInit:NOP   0;

      A     #PLCAlarms.ReqSendAlarm[1];
      O     #PLCAlarms.ReqSendAlarm[2];
      O     #PLCAlarms.ReqSendAlarm[3];
      O     #PLCAlarms.ReqSendAlarm[4];
      O     #PLCAlarms.ReqSendAlarm[5];
      O     #PLCAlarms.ReqSendAlarm[6];
      O     #PLCAlarms.ReqSendAlarm[7];
      O     #PLCAlarms.ReqSendAlarm[8];
      O     #PLCAlarms.ReqSendAlarm[9];
      O     #PLCAlarms.ReqSendAlarm[10];
      O     #PLCAlarms.ReqSendAlarm[11];
      O     #PLCAlarms.ReqSendAlarm[12];
      O     #PLCAlarms.ReqSendAlarm[13];
      O     #PLCAlarms.ReqSendAlarm[14];
      O     #PLCAlarms.ReqSendAlarm[15];
      O     #PLCAlarms.ReqSendAlarm[16];
      O     #PLCAlarms.ReqSendAlarm[17];
      O     #PLCAlarms.ReqSendAlarm[18];
      O     #PLCAlarms.ReqSendAlarm[19];
      O     #PLCAlarms.ReqSendAlarm[20];
      O     #PLCAlarms.ReqSendAlarm[21];
      O     #PLCAlarms.ReqSendAlarm[22];
      O     #PLCAlarms.ReqSendAlarm[23];
      O     #PLCAlarms.ReqSendAlarm[24];
      O     #PLCAlarms.ReqSendAlarm[25];
      O     #PLCAlarms.ReqSendAlarm[26];
      O     #PLCAlarms.ReqSendAlarm[27];
      O     #PLCAlarms.ReqSendAlarm[28];
      O     #PLCAlarms.ReqSendAlarm[29];
      O     #PLCAlarms.ReqSendAlarm[30];
      O     #PLCAlarms.ReqSendAlarm[31];
      O     #PLCAlarms.ReqSendAlarm[32];
      O     #PLCAlarms.ActiveRequest[1];
      O     #PLCAlarms.ActiveRequest[2];
      O     #PLCAlarms.ActiveRequest[3];
      O     #PLCAlarms.ActiveRequest[4];
      O     #PLCAlarms.ActiveRequest[5];
      O     #PLCAlarms.ActiveRequest[6];
      O     #PLCAlarms.ActiveRequest[7];
      O     #PLCAlarms.ActiveRequest[8];
      O     #PLCAlarms.ActiveRequest[9];
      O     #PLCAlarms.ActiveRequest[10];
      O     #PLCAlarms.ActiveRequest[11];
      O     #PLCAlarms.ActiveRequest[12];
      O     #PLCAlarms.ActiveRequest[13];
      O     #PLCAlarms.ActiveRequest[14];
      O     #PLCAlarms.ActiveRequest[15];
      O     #PLCAlarms.ActiveRequest[16];
      O     #PLCAlarms.ActiveRequest[17];
      O     #PLCAlarms.ActiveRequest[18];
      O     #PLCAlarms.ActiveRequest[19];
      O     #PLCAlarms.ActiveRequest[20];
      O     #PLCAlarms.ActiveRequest[21];
      O     #PLCAlarms.ActiveRequest[22];
      O     #PLCAlarms.ActiveRequest[23];
      O     #PLCAlarms.ActiveRequest[24];
      O     #PLCAlarms.ActiveRequest[25];
      O     #PLCAlarms.ActiveRequest[26];
      O     #PLCAlarms.ActiveRequest[27];
      O     #PLCAlarms.ActiveRequest[28];
      O     #PLCAlarms.ActiveRequest[29];
      O     #PLCAlarms.ActiveRequest[30];
      O     #PLCAlarms.ActiveRequest[31];
      O     #PLCAlarms.ActiveRequest[32];
      =     #InitUDT;


REGION Network 20: **** 4.4 - Machine status - Calculated ****Check Send Request
   // Check Send Request
   IF "TRUE" THEN "NotUsedInt" := BLKMOV(SRCBLK := #ReqSendToVDAlarm, DSTBLK => #ActiveRequest); END_IF;
END_REGION

REGION Network 21: **** 4.4 - Machine status - Calculated ****Check Send Done
   // Check Send Done
   IF "TRUE" THEN "NotUsedInt" := BLKMOV(SRCBLK := #SendAlarmDone, DSTBLK => #SendDoneArr); END_IF;
END_REGION

REGION Network 22: **** 4.4 - Machine status - Calculated ****Check Send Done
   // Check Send Done
   #_SendDoneReset(IN := (#SendDoneArr[0] <> DW#0) OR (#SendDoneArr[1] <> DW#0) OR #SendDoneVD OR #SendToVD OR #InitUDT,   // TON
                   PT := T#30s,
                   ET => "NotUsedTime");
   #ResetSendDone := #_SendDoneReset.Q;
END_REGION

REGION Network 23: **** 4.4 - Machine status - Calculated **** Ok To Request
   // Ok To Request
   #OkToRequest := (#ActiveRequest = DW#16#0000_0000) AND NOT #SendToVD AND NOT #SendDoneVD;
   IF #OkToRequest OR #SendDoneVD THEN #AlarmPointer := INT#0; END_IF;
END_REGION

REGION Network 24: **** 4.4 - Machine status - Calculated **** Delay Send To VD
   // Delay Send To VD
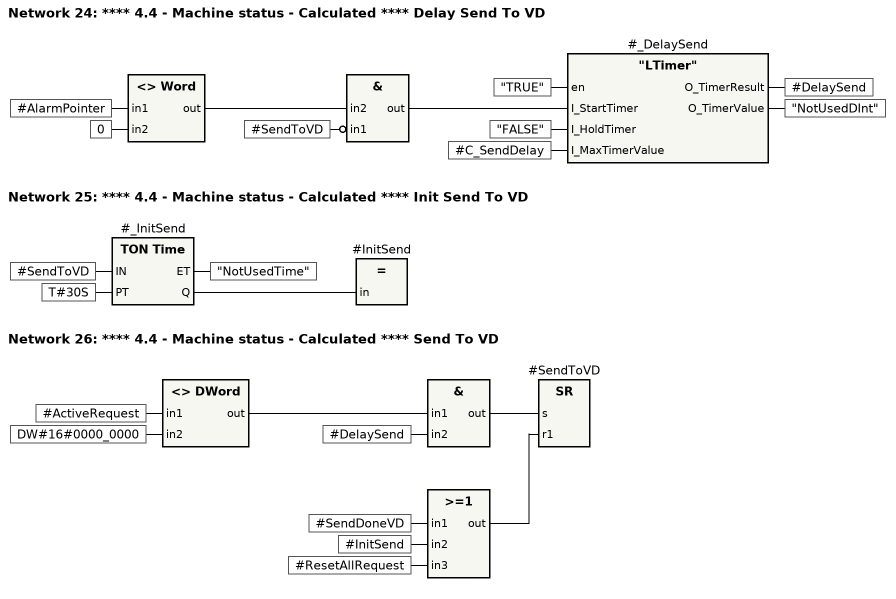
   IF "TRUE" THEN
       #_DelaySend(I_StartTimer := (#AlarmPointer <> 0) AND NOT #SendToVD,   // "LTimer"
                   I_HoldTimer := "FALSE",
                   I_MaxTimerValue := #C_SendDelay,
                   O_TimerResult => #DelaySend,
                   O_TimerValue => "NotUsedDInt");
   END_IF;
END_REGION

REGION Network 25: **** 4.4 - Machine status - Calculated **** Init Send To VD
   // Init Send To VD
   #_InitSend(IN := #SendToVD, PT := T#30S, ET => "NotUsedTime");   // TON
   #InitSend := #_InitSend.Q;
END_REGION

REGION Network 26: **** 4.4 - Machine status - Calculated **** Send To VD
   // Send To VD
   IF (#ActiveRequest <> DW#16#0000_0000) AND #DelaySend THEN
       #SendToVD := TRUE;   // SR flip-flop
   END_IF;
   IF #SendDoneVD OR #InitSend OR #ResetAllRequest THEN #SendToVD := FALSE; END_IF;
END_REGION

NETWORK
TITLE = **** 4.4 - Machine status - Calculated **** Header Send
// Header
// Configure Header For Send Data Alarm, APA// S7-1500 Preparations
      OPN   #C_LocalSendDB;
      L     DBNO;
      T     #SendDBBufNbr;
//    L     #AlarmPointer
//      T     #Pointer
//   OPN DB [ #Pointer]

//      T     #SendDBNbr
//    L DBLG
//  T     #AlarmLength
//
//    NOP 0
      L     #AlarmPointer;
      L     0;
      <>I;
      JCN   NozHeaD;
      L     #AlarmLength;
      +     10;
      T     #SendLength;

      LAR1  P##BPtr;
      L     16#1002;
      T     LW [AR1, P#0.0];
      L     #AlarmLength;
      T     LW [AR1, P#2.0];
      L     #AlarmPointer;
      T     LW [AR1, P#4.0];
      L     0;
      SLD   3;
      OD    16#8400_0000;
      T     LD [AR1, P#6.0];


      LAR1  P##SPtr;
      L     16#1002;
      T     LW [AR1, P#0.0];
      L     #AlarmLength;
      T     LW [AR1, P#2.0];
      L     #SendDBBufNbr;
      T     LW [AR1, P#4.0];
      L     10;
      SLD   3;
      OD    16#8400_0000;
      T     LD [AR1, P#6.0];
      CALL  BLKMOV
      ( SRCBLK  := #BPtr,
        RET_VAL := "NotUsedInt",
        DSTBLK  := #SPtr
      );
NozHeaD:NOP   0;


REGION Network 28: **** 5.2 - Equations - Flow Equations **** Header DB's
   // Header
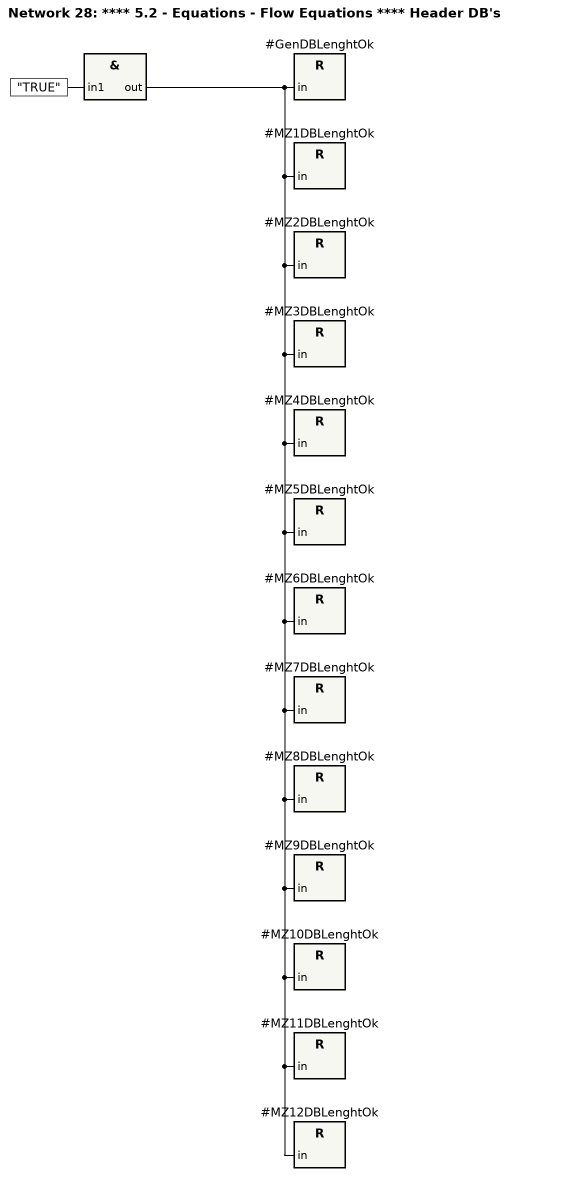
   IF "TRUE" THEN
       #GenDBLenghtOk := FALSE;
       #MZ1DBLenghtOk := FALSE;
       #MZ2DBLenghtOk := FALSE;
       #MZ3DBLenghtOk := FALSE;
       #MZ4DBLenghtOk := FALSE;
       #MZ5DBLenghtOk := FALSE;
       #MZ6DBLenghtOk := FALSE;
       #MZ7DBLenghtOk := FALSE;
       #MZ8DBLenghtOk := FALSE;
       #MZ9DBLenghtOk := FALSE;
       #MZ10DBLenghtOk := FALSE;
       #MZ11DBLenghtOk := FALSE;
       #MZ12DBLenghtOk := FALSE;
   END_IF;
END_REGION

NETWORK
TITLE = **** 5.2 - Equations - Flow Equations **** Header DB's
// Load Pointers For All Alarm DB:s


      OPN   #C_GenAlarmDB;  //General PLC Alarms
      L     DBLG;
      T     %DBW0;
      T     #GenDBLength;
      L     DBNO;
      T     #GenDBNumber;
      T     %DBW2;
      OPN   #C_GenAlarmCompare;  //General PLC Alarms
      L     DBLG;
      T     #GenDBLenghtCompare;
      L     #GenDBLength;
      L     #GenDBLenghtCompare;
      ==D;
      JCN   GenOk;
      L     #GenDBLenghtCompare;
      L     8;
      >=I;
      S     #GenDBLenghtOk;
GenOk:NOP   0;
      OPN   #C_AlarmDBMZ1;  // MZ Alarms
      L     DBLG;
      T     %DBW0;
      T     #MZ1DBLength;
      L     DBNO;
      T     #MZ1DBNumber;
      T     %DBW2;
      OPN   #C_AlarmCompareDBMZ1;  //MZ Alarms
      L     DBLG;
      T     #MZ1DBLenghtCompare;
      L     #MZ1DBLength;
      L     #MZ1DBLenghtCompare;
      ==D;
      JCN   MZ1Ok;
      L     #MZ1DBLenghtCompare;
      L     8;
      >=I;
      S     #MZ1DBLenghtOk;
MZ1Ok:NOP   0;
      OPN   #C_AlarmDBMZ2;  // MZ Alarms
      L     DBLG;
      T     %DBW0;
      T     #MZ2DBLength;
      L     DBNO;
      T     #MZ2DBNumber;
      T     %DBW2;
      OPN   #C_AlarmCompareDBMZ2;  //MZ Alarms
      L     DBLG;
      T     #MZ2DBLenghtCompare;
      L     #MZ2DBLength;
      L     #MZ2DBLenghtCompare;
      ==D;
      JCN   MZ2ok;
      L     #MZ2DBLenghtCompare;
      L     8;
      >=I;
      S     #MZ2DBLenghtOk;
MZ2ok:NOP   0;
      OPN   #C_AlarmDBMZ3;  // MZ Alarms
      L     DBLG;
      T     %DBW0;
      T     #MZ3DBLength;
      L     DBNO;
      T     #MZ3DBNumber;
      T     %DBW2;
      OPN   #C_AlarmCompareDBMZ3;  //MZ Alarms
      L     DBLG;
      T     #MZ3DBLenghtCompare;
      L     #MZ3DBLength;
      L     #MZ3DBLenghtCompare;
      ==D;
      JCN   MZ3ok;
      L     #MZ3DBLenghtCompare;
      L     8;
      >=I;
      S     #MZ3DBLenghtOk;
MZ3ok:NOP   0;
      OPN   #C_AlarmDBMZ4;  // MZ Alarms
      L     DBLG;
      T     %DBW0;
      T     #MZ4DBLength;
      L     DBNO;
      T     #MZ4DBNumber;
      T     %DBW2;
      OPN   #C_AlarmCompareDBMZ4;  //MZ Alarms
      L     DBLG;
      T     #MZ4DBLenghtCompare;
      L     #MZ4DBLength;
      L     #MZ4DBLenghtCompare;
      ==D;
      JCN   MZ4ok;
      L     #MZ4DBLenghtCompare;
      L     8;
      >=I;
      S     #MZ4DBLenghtOk;
MZ4ok:NOP   0;
      OPN   #C_AlarmDBMZ5;  // MZ Alarms
      L     DBLG;
      T     %DBW0;
      T     #MZ5DBLength;
      L     DBNO;
      T     #MZ5DBNumber;
      T     %DBW2;
      OPN   #C_AlarmCompareDBMZ5;  //MZ Alarms
      L     DBLG;
      T     #MZ5DBLenghtCompare;
      L     #MZ5DBLength;
      L     #MZ5DBLenghtCompare;
      ==D;
      JCN   MZ5ok;
      L     #MZ5DBLenghtCompare;
      L     8;
      >=I;
      S     #MZ5DBLenghtOk;
MZ5ok:NOP   0;
      OPN   #C_AlarmDBMZ6;  // MZ Alarms
      L     DBLG;
      T     %DBW0;
      T     #MZ6DBLength;
      L     DBNO;
      T     #MZ6DBNumber;
      T     %DBW2;
      OPN   #C_AlarmCompareDBMZ6;  //MZ Alarms
      L     DBLG;
      T     #MZ6DBLenghtCompare;
      L     #MZ6DBLength;
      L     #MZ6DBLenghtCompare;
      ==D;
      JCN   MZ6ok;
      L     #MZ6DBLenghtCompare;
      L     8;
      >=I;
      S     #MZ6DBLenghtOk;
MZ6ok:NOP   0;
      OPN   #C_AlarmDBMZ7;  // MZ Alarms
      L     DBLG;
      T     %DBW0;
      T     #MZ7DBLength;
      L     DBNO;
      T     #MZ7DBNumber;
      T     %DBW2;
      OPN   #C_AlarmCompareDBMZ7;  //MZ Alarms
      L     DBLG;
      T     #MZ7DBLenghtCompare;
      L     #MZ7DBLength;
      L     #MZ7DBLenghtCompare;
      ==D;
      JCN   MZ7ok;
      L     #MZ7DBLenghtCompare;
      L     8;
      >=I;
      S     #MZ7DBLenghtOk;
MZ7ok:NOP   0;
      OPN   #C_AlarmDBMZ8;  // MZ Alarms
      L     DBLG;
      T     %DBW0;
      T     #MZ8DBLength;
      L     DBNO;
      T     #MZ8DBNumber;
      T     %DBW2;
      OPN   #C_AlarmCompareDBMZ8;  //MZ Alarms
      L     DBLG;
      T     #MZ8DBLenghtCompare;
      L     #MZ8DBLength;
      L     #MZ8DBLenghtCompare;
      ==D;
      JCN   MZ8ok;
      L     #MZ8DBLenghtCompare;
      L     8;
      >=I;
      S     #MZ8DBLenghtOk;
MZ8ok:NOP   0;
      OPN   #C_AlarmDBMZ9;  // MZ Alarms
      L     DBLG;
      T     %DBW0;
      T     #MZ9DBLength;
      L     DBNO;
      T     #MZ9DBNumber;
      T     %DBW2;
      OPN   #C_AlarmCompareDBMZ9;  //MZ Alarms
      L     DBLG;
      T     #MZ9DBLenghtCompare;
      L     #MZ9DBLength;
      L     #MZ9DBLenghtCompare;
      ==D;
      JCN   MZ9ok;
      L     #MZ9DBLenghtCompare;
      L     8;
      >=I;
      S     #MZ9DBLenghtOk;
MZ9ok:NOP   0;
      OPN   #C_AlarmDBMZ10;  // MZ Alarms
      L     DBLG;
      T     %DBW0;
      T     #MZ10DBLength;
      L     DBNO;
      T     #MZ10DBNumber;
      T     %DBW2;
      OPN   #C_AlarmCompareDBMZ10;  //MZ Alarms
      L     DBLG;
      T     #MZ10DBLenghtCompare;
      L     #MZ10DBLength;
      L     #MZ10DBLenghtCompare;
      ==D;
      JCN   MZ10ok;
      L     #MZ10DBLenghtCompare;
      L     8;
      >=I;
      S     #MZ10DBLenghtOk;
MZ10ok:NOP   0;
      OPN   #C_AlarmDBMZ11;  // MZ Alarms
      L     DBLG;
      T     %DBW0;
      T     #MZ11DBLength;
      L     DBNO;
      T     #MZ11DBNumber;
      T     %DBW2;
      OPN   #C_AlarmCompareDBMZ11;  //MZ Alarms
      L     DBLG;
      T     #MZ11DBLenghtCompare;
      L     #MZ11DBLength;
      L     #MZ11DBLenghtCompare;
      ==D;
      JCN   MZ11ok;
      L     #MZ11DBLenghtCompare;
      L     8;
      >=I;
      S     #MZ11DBLenghtOk;
MZ11ok:NOP   0;
      OPN   #C_AlarmDBMZ12;  // MZ Alarms
      L     DBLG;
      T     %DBW0;
      T     #MZ12DBLength;
      L     DBNO;
      T     #MZ12DBNumber;
      OPN   #C_AlarmCompareDBMZ12;  //MZ Alarms
      L     DBLG;
      T     #MZ12DBLenghtCompare;
      L     #MZ12DBLength;
      L     #MZ12DBLenghtCompare;
      ==D;
      JCN   MZ12ok;
      L     #MZ12DBLenghtCompare;
      L     8;
      >=I;
      S     #MZ12DBLenghtOk;
MZ12ok:NOP   0;

      OPN   #C_AlarmDBMZ13;  // MZ Alarms
      L     DBLG;
      T     %DBW0;
      T     #MZ13DBLength;
      L     DBNO;
      T     #MZ13DBNumber;
      OPN   #C_AlarmCompareDBMZ13;  //MZ Alarms
      L     DBLG;
      T     #MZ13DBLenghtCompare;
      L     #MZ13DBLength;
      L     #MZ13DBLenghtCompare;
      ==D;
      JCN   MZ13ok;
      L     #MZ13DBLenghtCompare;
      L     8;
      >=I;
      S     #MZ13DBLenghtOk;

MZ13ok:NOP   0;

      OPN   #C_AlarmDBMZ14;  // MZ Alarms
      L     DBLG;
      T     %DBW0;
      T     #MZ14DBLength;
      L     DBNO;
      T     #MZ14DBNumber;
      OPN   #C_AlarmCompareDBMZ14;  //MZ Alarms
      L     DBLG;
      T     #MZ14DBLenghtCompare;
      L     #MZ14DBLength;
      L     #MZ14DBLenghtCompare;
      ==D;
      JCN   MZ14ok;
      L     #MZ14DBLenghtCompare;
      L     8;
      >=I;
      S     #MZ14DBLenghtOk;

MZ14ok:NOP   0;

//Alarm DB's Ok To Send
      A     #GenDBLenghtOk;
      =     #IO_AlarmDB.GenDBLenghtOk;
      A     #MZ1DBLenghtOk;
      =     #IO_AlarmDB.MZ1DBLenghtOk;
      A     #MZ2DBLenghtOk;
      =     #IO_AlarmDB.MZ2DBLenghtOk;
      A     #MZ3DBLenghtOk;
      =     #IO_AlarmDB.MZ3DBLenghtOk;
      A     #MZ4DBLenghtOk;
      =     #IO_AlarmDB.MZ4DBLenghtOk;
      A     #MZ5DBLenghtOk;
      =     #IO_AlarmDB.MZ5DBLenghtOk;
      A     #MZ6DBLenghtOk;
      =     #IO_AlarmDB.MZ6DBLenghtOk;
      A     #MZ7DBLenghtOk;
      =     #IO_AlarmDB.MZ7DBLenghtOk;
      A     #MZ8DBLenghtOk;
      =     #IO_AlarmDB.MZ8DBLenghtOk;
      A     #MZ9DBLenghtOk;
      =     #IO_AlarmDB.MZ9DBLenghtOk;
      A     #MZ10DBLenghtOk;
      =     #IO_AlarmDB.MZ10DBLenghtOk;
      A     #MZ11DBLenghtOk;
      =     #IO_AlarmDB.MZ11DBLenghtOk;
      A     #MZ12DBLenghtOk;
      =     #IO_AlarmDB.MZ12DBLenghtOk;
      A     #MZ13DBLenghtOk;
      =     #IO_AlarmDB.MZ13DBLenghtOk;
      A     #MZ14DBLenghtOk;
      =     #IO_AlarmDB.MZ14DBLenghtOk;

// Amount Of ModeZone
      L     #C_NbrOfModeZone;
      T     #IO_AlarmDB.C_NbrOfModeZone;


REGION Network 30: **** 5.2 - Flow Equations **** Filter
   // Filter
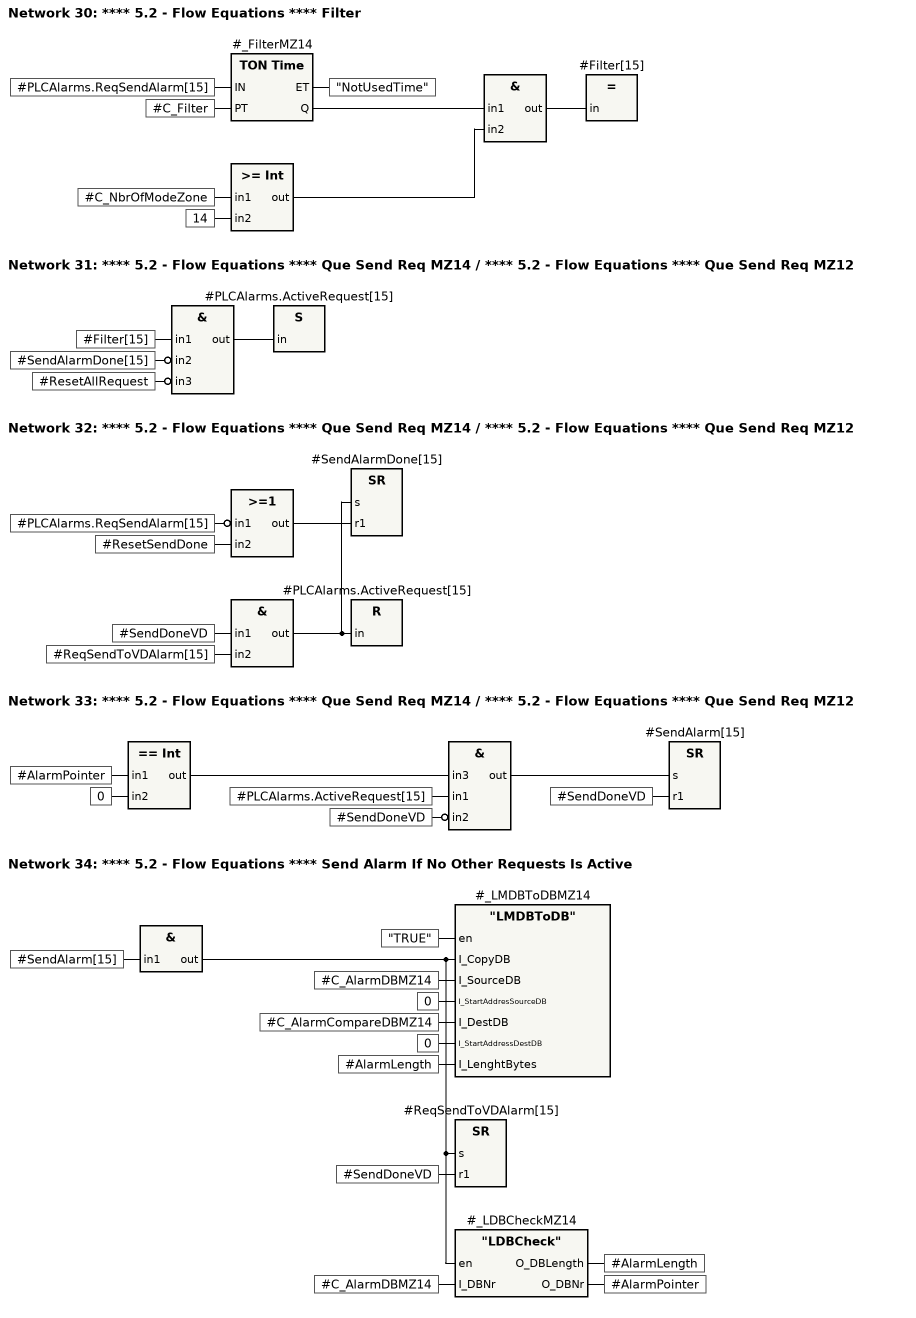
   #_FilterMZ14(IN := #PLCAlarms.ReqSendAlarm[15], PT := #C_Filter, ET => "NotUsedTime");   // TON
   #Filter[15] := #_FilterMZ14.Q AND (#C_NbrOfModeZone >= 14);
END_REGION

REGION Network 31: **** 5.2 - Flow Equations **** Que Send Req MZ14 / **** 5.2 - Flow Equations **** Que Send Req MZ12
   // Que Send Req
   IF #Filter[15] AND NOT #SendAlarmDone[15] AND NOT #ResetAllRequest THEN
       #PLCAlarms.ActiveRequest[15] := TRUE;
   END_IF;
END_REGION

REGION Network 32: **** 5.2 - Flow Equations **** Que Send Req MZ14 / **** 5.2 - Flow Equations **** Que Send Req MZ12
   // Que Send Req
   #_w1 := #SendDoneVD AND #ReqSendToVDAlarm[15];
   IF #_w1 THEN
       #SendAlarmDone[15] := TRUE;   // SR flip-flop
   END_IF;
   IF NOT #PLCAlarms.ReqSendAlarm[15] OR #ResetSendDone THEN #SendAlarmDone[15] := FALSE; END_IF;
   IF #_w1 THEN #PLCAlarms.ActiveRequest[15] := FALSE; END_IF;
END_REGION

REGION Network 33: **** 5.2 - Flow Equations **** Que Send Req MZ14 / **** 5.2 - Flow Equations **** Que Send Req MZ12
   // Que Send Req
   IF (#AlarmPointer = 0) AND #PLCAlarms.ActiveRequest[15] AND NOT #SendDoneVD THEN
       #SendAlarm[15] := TRUE;   // SR flip-flop
   END_IF;
   IF #SendDoneVD THEN #SendAlarm[15] := FALSE; END_IF;
END_REGION

REGION Network 34: **** 5.2 - Flow Equations **** Send Alarm If No Other Requests Is Active
   // Send Alarm If No Other Requests Is Active
   IF #SendAlarm[15] THEN
       #ReqSendToVDAlarm[15] := TRUE;   // SR flip-flop
   END_IF;
   IF #SendDoneVD THEN #ReqSendToVDAlarm[15] := FALSE; END_IF;
   IF #SendAlarm[15] THEN
       #_LDBCheckMZ14(I_DBNr := #C_AlarmDBMZ14, O_DBLength => #AlarmLength, O_DBNr => #AlarmPointer);   // "LDBCheck"
   END_IF;
   IF "TRUE" THEN
       #_LMDBToDBMZ14(I_CopyDB := #SendAlarm[15],   // "LMDBToDB"
                      I_SourceDB := #C_AlarmDBMZ14,
                      I_StartAddresSourceDB := 0,
                      I_DestDB := #C_AlarmCompareDBMZ14,
                      I_StartAddressDestDB := 0,
                      I_LenghtBytes := #AlarmLength);
   END_IF;
END_REGION

REGION Network 35: **** 5.2 - Flow Equations **** Filter
   // Filter
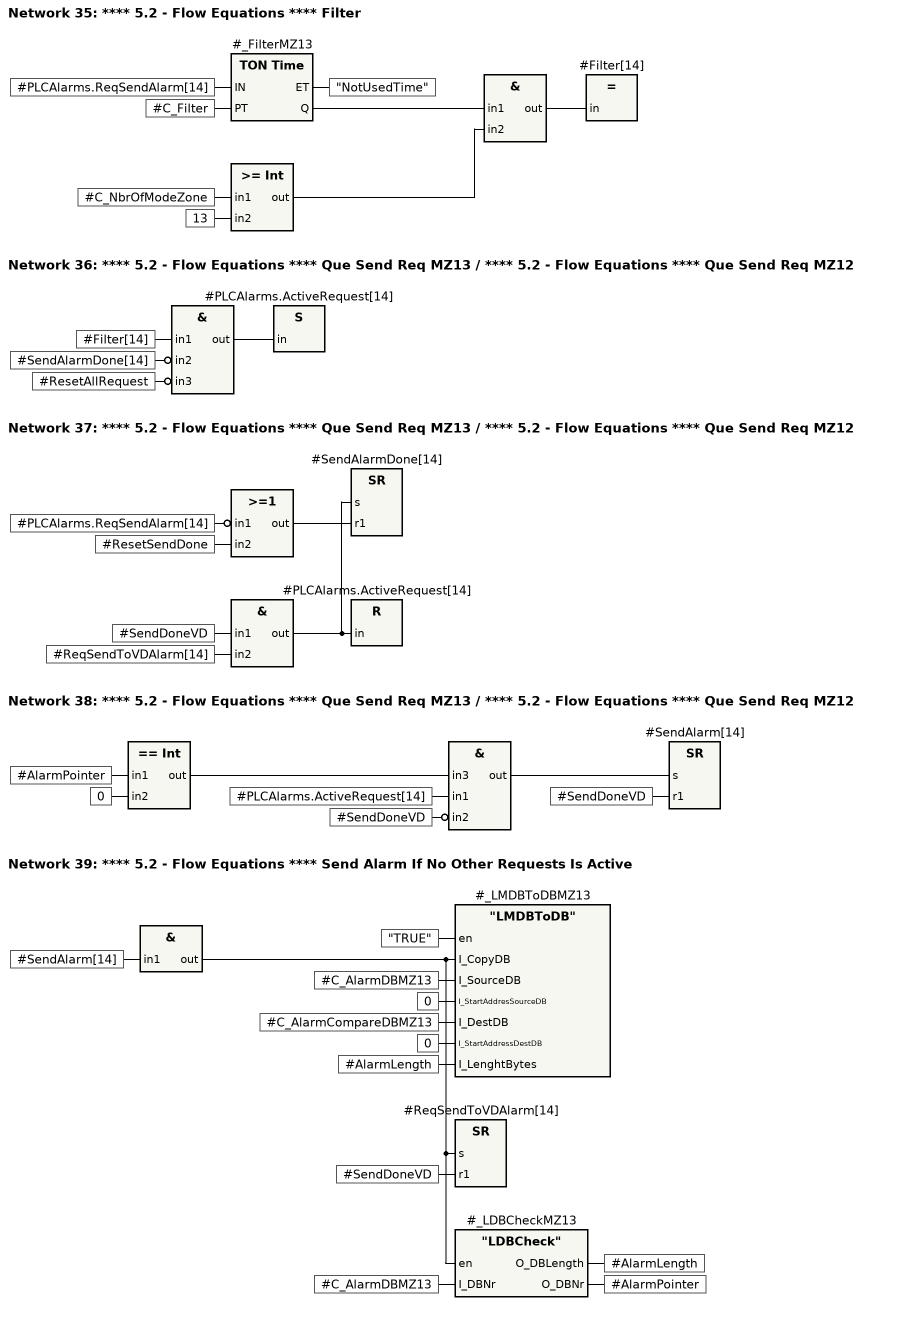
   #_FilterMZ13(IN := #PLCAlarms.ReqSendAlarm[14], PT := #C_Filter, ET => "NotUsedTime");   // TON
   #Filter[14] := #_FilterMZ13.Q AND (#C_NbrOfModeZone >= 13);
END_REGION

REGION Network 36: **** 5.2 - Flow Equations **** Que Send Req MZ13 / **** 5.2 - Flow Equations **** Que Send Req MZ12
   // Que Send Req
   IF #Filter[14] AND NOT #SendAlarmDone[14] AND NOT #ResetAllRequest THEN
       #PLCAlarms.ActiveRequest[14] := TRUE;
   END_IF;
END_REGION

REGION Network 37: **** 5.2 - Flow Equations **** Que Send Req MZ13 / **** 5.2 - Flow Equations **** Que Send Req MZ12
   // Que Send Req
   #_w1 := #SendDoneVD AND #ReqSendToVDAlarm[14];
   IF #_w1 THEN
       #SendAlarmDone[14] := TRUE;   // SR flip-flop
   END_IF;
   IF NOT #PLCAlarms.ReqSendAlarm[14] OR #ResetSendDone THEN #SendAlarmDone[14] := FALSE; END_IF;
   IF #_w1 THEN #PLCAlarms.ActiveRequest[14] := FALSE; END_IF;
END_REGION

REGION Network 38: **** 5.2 - Flow Equations **** Que Send Req MZ13 / **** 5.2 - Flow Equations **** Que Send Req MZ12
   // Que Send Req
   IF (#AlarmPointer = 0) AND #PLCAlarms.ActiveRequest[14] AND NOT #SendDoneVD THEN
       #SendAlarm[14] := TRUE;   // SR flip-flop
   END_IF;
   IF #SendDoneVD THEN #SendAlarm[14] := FALSE; END_IF;
END_REGION

REGION Network 39: **** 5.2 - Flow Equations **** Send Alarm If No Other Requests Is Active
   // Send Alarm If No Other Requests Is Active
   IF #SendAlarm[14] THEN
       #ReqSendToVDAlarm[14] := TRUE;   // SR flip-flop
   END_IF;
   IF #SendDoneVD THEN #ReqSendToVDAlarm[14] := FALSE; END_IF;
   IF #SendAlarm[14] THEN
       #_LDBCheckMZ13(I_DBNr := #C_AlarmDBMZ13, O_DBLength => #AlarmLength, O_DBNr => #AlarmPointer);   // "LDBCheck"
   END_IF;
   IF "TRUE" THEN
       #_LMDBToDBMZ13(I_CopyDB := #SendAlarm[14],   // "LMDBToDB"
                      I_SourceDB := #C_AlarmDBMZ13,
                      I_StartAddresSourceDB := 0,
                      I_DestDB := #C_AlarmCompareDBMZ13,
                      I_StartAddressDestDB := 0,
                      I_LenghtBytes := #AlarmLength);
   END_IF;
END_REGION

REGION Network 40: **** 5.2 - Flow Equations **** Filter
   // Filter
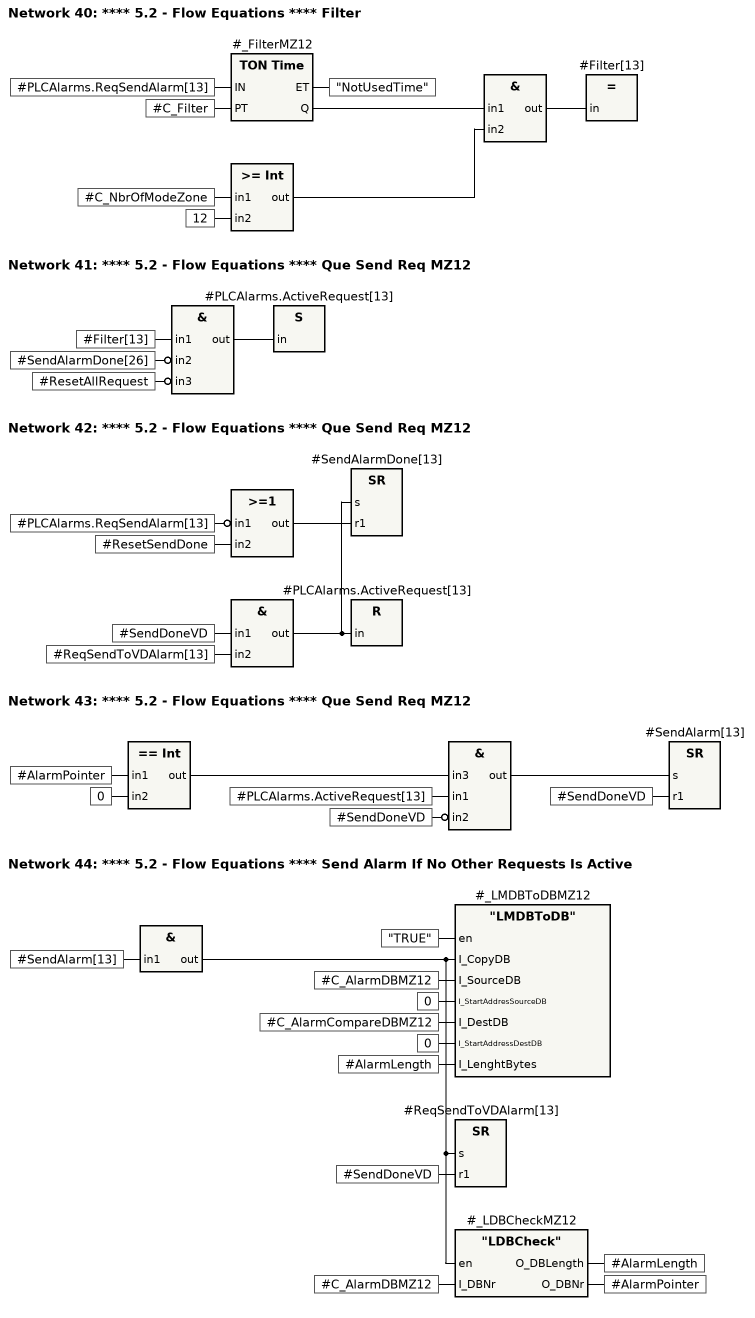
   #_FilterMZ12(IN := #PLCAlarms.ReqSendAlarm[13], PT := #C_Filter, ET => "NotUsedTime");   // TON
   #Filter[13] := #_FilterMZ12.Q AND (#C_NbrOfModeZone >= 12);
END_REGION

REGION Network 41: **** 5.2 - Flow Equations **** Que Send Req MZ12
   // Que Send Req
   IF #Filter[13] AND NOT #SendAlarmDone[26] AND NOT #ResetAllRequest THEN
       #PLCAlarms.ActiveRequest[13] := TRUE;
   END_IF;
END_REGION

REGION Network 42: **** 5.2 - Flow Equations **** Que Send Req MZ12
   // Que Send Req
   #_w1 := #SendDoneVD AND #ReqSendToVDAlarm[13];
   IF #_w1 THEN
       #SendAlarmDone[13] := TRUE;   // SR flip-flop
   END_IF;
   IF NOT #PLCAlarms.ReqSendAlarm[13] OR #ResetSendDone THEN #SendAlarmDone[13] := FALSE; END_IF;
   IF #_w1 THEN #PLCAlarms.ActiveRequest[13] := FALSE; END_IF;
END_REGION

REGION Network 43: **** 5.2 - Flow Equations **** Que Send Req MZ12
   // Que Send Req
   IF (#AlarmPointer = 0) AND #PLCAlarms.ActiveRequest[13] AND NOT #SendDoneVD THEN
       #SendAlarm[13] := TRUE;   // SR flip-flop
   END_IF;
   IF #SendDoneVD THEN #SendAlarm[13] := FALSE; END_IF;
END_REGION

REGION Network 44: **** 5.2 - Flow Equations **** Send Alarm If No Other Requests Is Active
   // Send Alarm If No Other Requests Is Active
   IF #SendAlarm[13] THEN
       #ReqSendToVDAlarm[13] := TRUE;   // SR flip-flop
   END_IF;
   IF #SendDoneVD THEN #ReqSendToVDAlarm[13] := FALSE; END_IF;
   IF #SendAlarm[13] THEN
       #_LDBCheckMZ12(I_DBNr := #C_AlarmDBMZ12, O_DBLength => #AlarmLength, O_DBNr => #AlarmPointer);   // "LDBCheck"
   END_IF;
   IF "TRUE" THEN
       #_LMDBToDBMZ12(I_CopyDB := #SendAlarm[13],   // "LMDBToDB"
                      I_SourceDB := #C_AlarmDBMZ12,
                      I_StartAddresSourceDB := 0,
                      I_DestDB := #C_AlarmCompareDBMZ12,
                      I_StartAddressDestDB := 0,
                      I_LenghtBytes := #AlarmLength);
   END_IF;
END_REGION

REGION Network 45: **** 5.2 - Flow Equations **** Filter
   // Filter
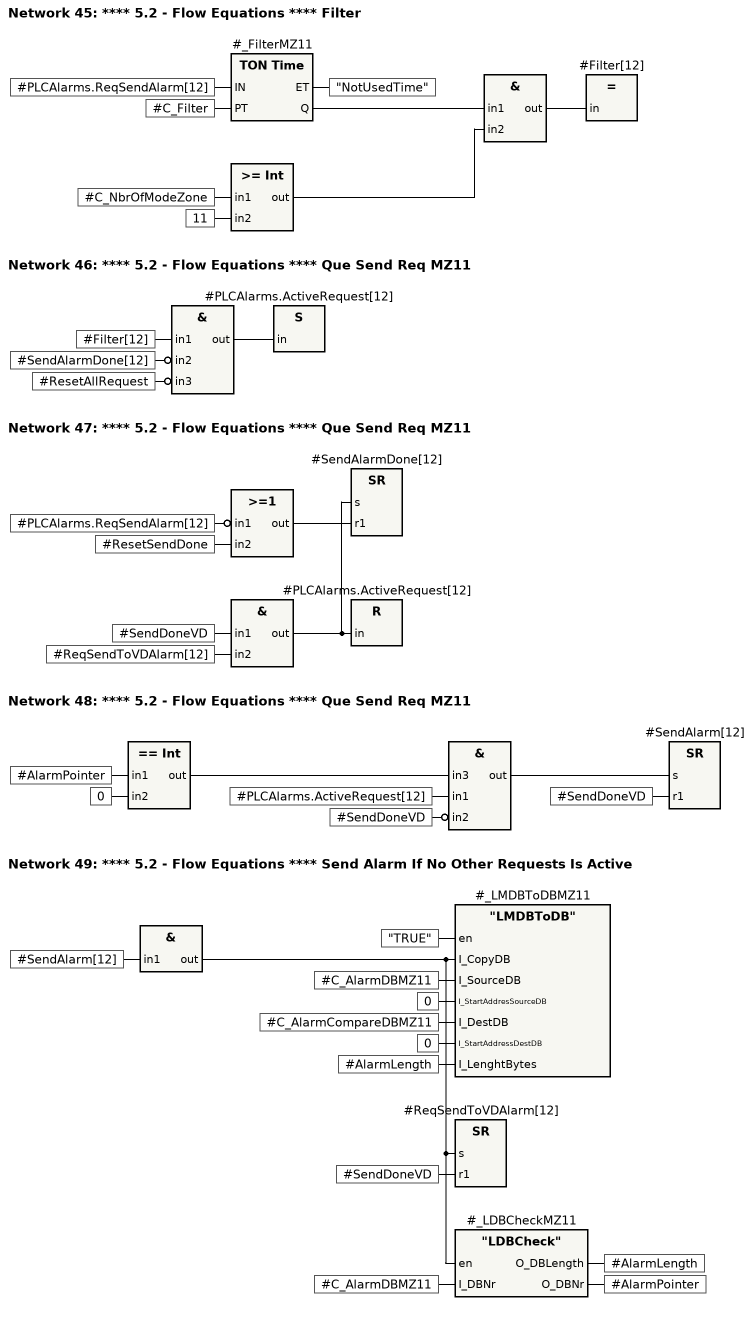
   #_FilterMZ11(IN := #PLCAlarms.ReqSendAlarm[12], PT := #C_Filter, ET => "NotUsedTime");   // TON
   #Filter[12] := #_FilterMZ11.Q AND (#C_NbrOfModeZone >= 11);
END_REGION

REGION Network 46: **** 5.2 - Flow Equations **** Que Send Req MZ11
   // Que Send Req
   IF #Filter[12] AND NOT #SendAlarmDone[12] AND NOT #ResetAllRequest THEN
       #PLCAlarms.ActiveRequest[12] := TRUE;
   END_IF;
END_REGION

REGION Network 47: **** 5.2 - Flow Equations **** Que Send Req MZ11
   // Que Send Req
   #_w1 := #SendDoneVD AND #ReqSendToVDAlarm[12];
   IF #_w1 THEN
       #SendAlarmDone[12] := TRUE;   // SR flip-flop
   END_IF;
   IF NOT #PLCAlarms.ReqSendAlarm[12] OR #ResetSendDone THEN #SendAlarmDone[12] := FALSE; END_IF;
   IF #_w1 THEN #PLCAlarms.ActiveRequest[12] := FALSE; END_IF;
END_REGION

REGION Network 48: **** 5.2 - Flow Equations **** Que Send Req MZ11
   // Que Send Req
   IF (#AlarmPointer = 0) AND #PLCAlarms.ActiveRequest[12] AND NOT #SendDoneVD THEN
       #SendAlarm[12] := TRUE;   // SR flip-flop
   END_IF;
   IF #SendDoneVD THEN #SendAlarm[12] := FALSE; END_IF;
END_REGION

REGION Network 49: **** 5.2 - Flow Equations **** Send Alarm If No Other Requests Is Active
   // Send Alarm If No Other Requests Is Active
   IF #SendAlarm[12] THEN
       #ReqSendToVDAlarm[12] := TRUE;   // SR flip-flop
   END_IF;
   IF #SendDoneVD THEN #ReqSendToVDAlarm[12] := FALSE; END_IF;
   IF #SendAlarm[12] THEN
       #_LDBCheckMZ11(I_DBNr := #C_AlarmDBMZ11, O_DBLength => #AlarmLength, O_DBNr => #AlarmPointer);   // "LDBCheck"
   END_IF;
   IF "TRUE" THEN
       #_LMDBToDBMZ11(I_CopyDB := #SendAlarm[12],   // "LMDBToDB"
                      I_SourceDB := #C_AlarmDBMZ11,
                      I_StartAddresSourceDB := 0,
                      I_DestDB := #C_AlarmCompareDBMZ11,
                      I_StartAddressDestDB := 0,
                      I_LenghtBytes := #AlarmLength);
   END_IF;
END_REGION

REGION Network 50: **** 5.2 - Flow Equations **** Filter
   // Filter
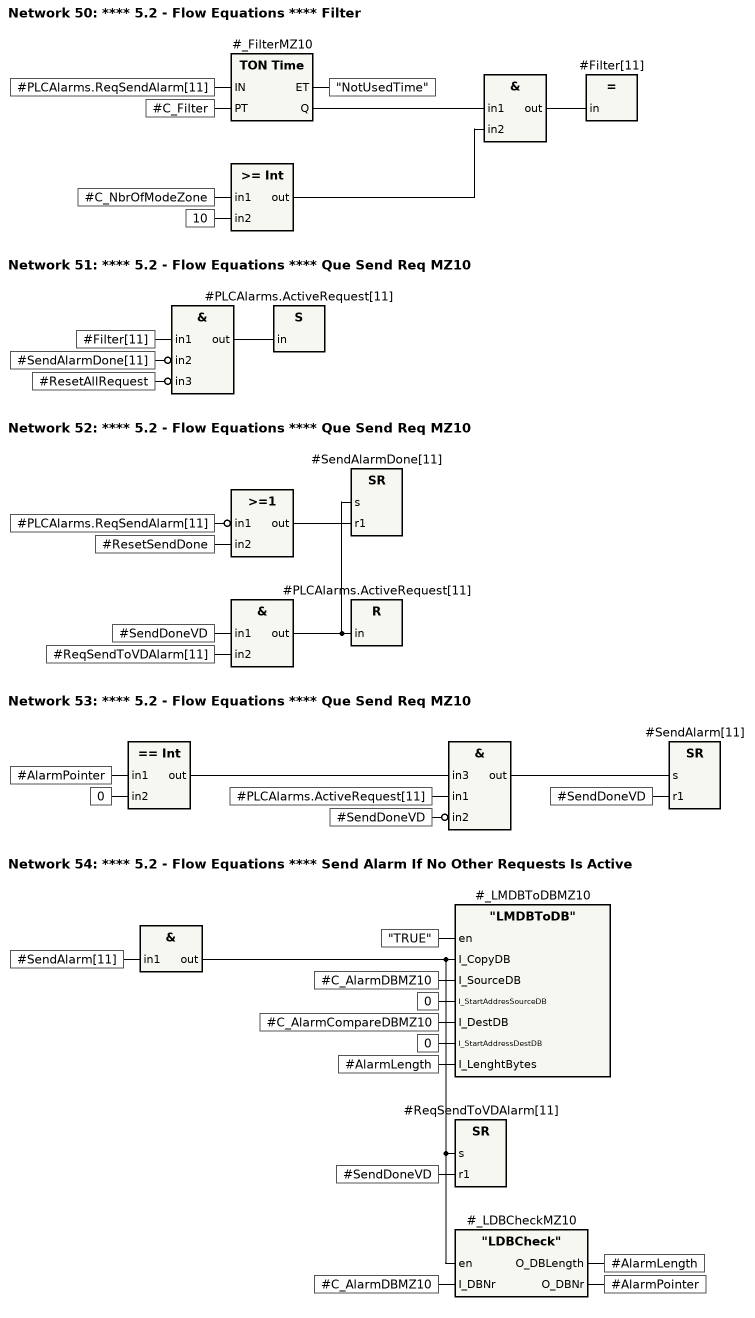
   #_FilterMZ10(IN := #PLCAlarms.ReqSendAlarm[11], PT := #C_Filter, ET => "NotUsedTime");   // TON
   #Filter[11] := #_FilterMZ10.Q AND (#C_NbrOfModeZone >= 10);
END_REGION

REGION Network 51: **** 5.2 - Flow Equations **** Que Send Req MZ10
   // Que Send Req
   IF #Filter[11] AND NOT #SendAlarmDone[11] AND NOT #ResetAllRequest THEN
       #PLCAlarms.ActiveRequest[11] := TRUE;
   END_IF;
END_REGION

REGION Network 52: **** 5.2 - Flow Equations **** Que Send Req MZ10
   // Que Send Req
   #_w1 := #SendDoneVD AND #ReqSendToVDAlarm[11];
   IF #_w1 THEN
       #SendAlarmDone[11] := TRUE;   // SR flip-flop
   END_IF;
   IF NOT #PLCAlarms.ReqSendAlarm[11] OR #ResetSendDone THEN #SendAlarmDone[11] := FALSE; END_IF;
   IF #_w1 THEN #PLCAlarms.ActiveRequest[11] := FALSE; END_IF;
END_REGION

REGION Network 53: **** 5.2 - Flow Equations **** Que Send Req MZ10
   // Que Send Req
   IF (#AlarmPointer = 0) AND #PLCAlarms.ActiveRequest[11] AND NOT #SendDoneVD THEN
       #SendAlarm[11] := TRUE;   // SR flip-flop
   END_IF;
   IF #SendDoneVD THEN #SendAlarm[11] := FALSE; END_IF;
END_REGION

REGION Network 54: **** 5.2 - Flow Equations **** Send Alarm If No Other Requests Is Active
   // Send Alarm If No Other Requests Is Active
   IF #SendAlarm[11] THEN
       #ReqSendToVDAlarm[11] := TRUE;   // SR flip-flop
   END_IF;
   IF #SendDoneVD THEN #ReqSendToVDAlarm[11] := FALSE; END_IF;
   IF #SendAlarm[11] THEN
       #_LDBCheckMZ10(I_DBNr := #C_AlarmDBMZ10, O_DBLength => #AlarmLength, O_DBNr => #AlarmPointer);   // "LDBCheck"
   END_IF;
   IF "TRUE" THEN
       #_LMDBToDBMZ10(I_CopyDB := #SendAlarm[11],   // "LMDBToDB"
                      I_SourceDB := #C_AlarmDBMZ10,
                      I_StartAddresSourceDB := 0,
                      I_DestDB := #C_AlarmCompareDBMZ10,
                      I_StartAddressDestDB := 0,
                      I_LenghtBytes := #AlarmLength);
   END_IF;
END_REGION

REGION Network 55: **** 5.2 - Flow Equations **** Filter
   // Filter
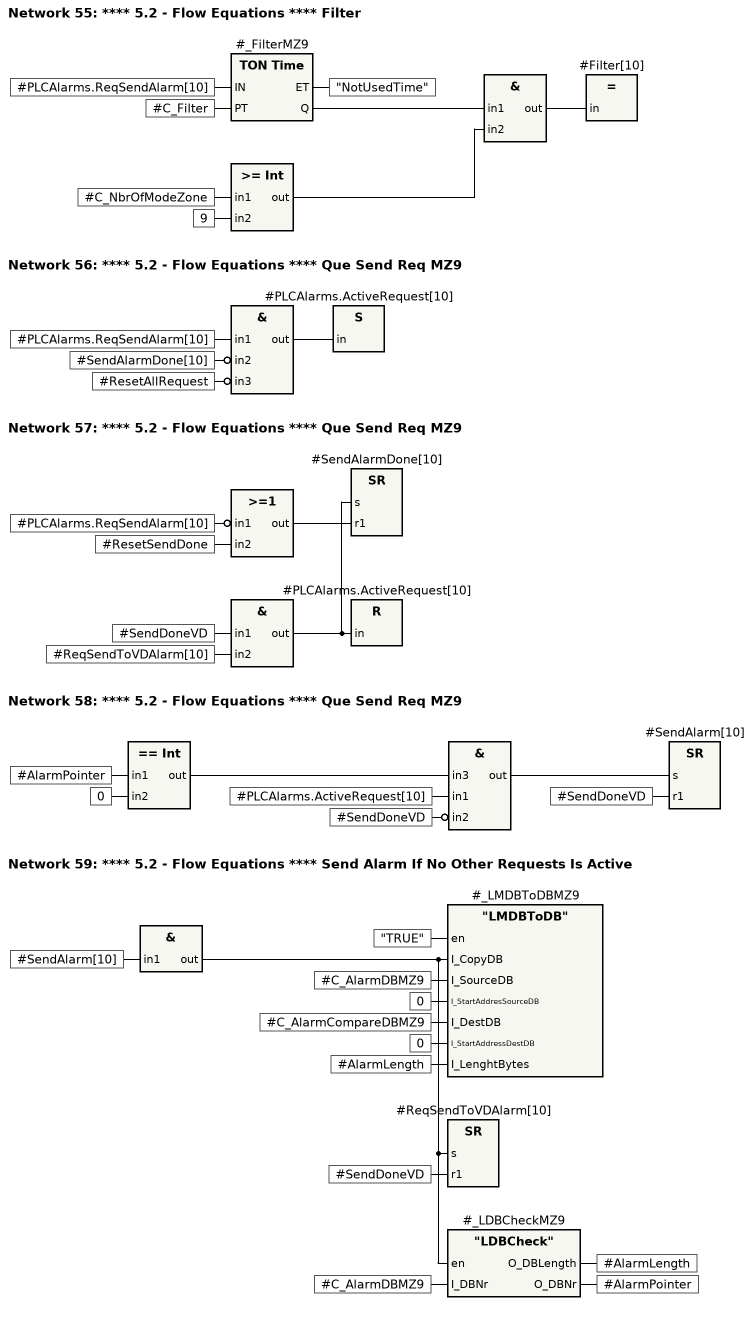
   #_FilterMZ9(IN := #PLCAlarms.ReqSendAlarm[10], PT := #C_Filter, ET => "NotUsedTime");   // TON
   #Filter[10] := #_FilterMZ9.Q AND (#C_NbrOfModeZone >= 9);
END_REGION

REGION Network 56: **** 5.2 - Flow Equations **** Que Send Req MZ9
   // Que Send Req
   IF #PLCAlarms.ReqSendAlarm[10] AND NOT #SendAlarmDone[10] AND NOT #ResetAllRequest THEN
       #PLCAlarms.ActiveRequest[10] := TRUE;
   END_IF;
END_REGION

REGION Network 57: **** 5.2 - Flow Equations **** Que Send Req MZ9
   // Que Send Req
   #_w1 := #SendDoneVD AND #ReqSendToVDAlarm[10];
   IF #_w1 THEN
       #SendAlarmDone[10] := TRUE;   // SR flip-flop
   END_IF;
   IF NOT #PLCAlarms.ReqSendAlarm[10] OR #ResetSendDone THEN #SendAlarmDone[10] := FALSE; END_IF;
   IF #_w1 THEN #PLCAlarms.ActiveRequest[10] := FALSE; END_IF;
END_REGION

REGION Network 58: **** 5.2 - Flow Equations **** Que Send Req MZ9
   // Que Send Req
   IF (#AlarmPointer = 0) AND #PLCAlarms.ActiveRequest[10] AND NOT #SendDoneVD THEN
       #SendAlarm[10] := TRUE;   // SR flip-flop
   END_IF;
   IF #SendDoneVD THEN #SendAlarm[10] := FALSE; END_IF;
END_REGION

REGION Network 59: **** 5.2 - Flow Equations **** Send Alarm If No Other Requests Is Active
   // Send Alarm If No Other Requests Is Active
   IF #SendAlarm[10] THEN
       #ReqSendToVDAlarm[10] := TRUE;   // SR flip-flop
   END_IF;
   IF #SendDoneVD THEN #ReqSendToVDAlarm[10] := FALSE; END_IF;
   IF #SendAlarm[10] THEN
       #_LDBCheckMZ9(I_DBNr := #C_AlarmDBMZ9, O_DBLength => #AlarmLength, O_DBNr => #AlarmPointer);   // "LDBCheck"
   END_IF;
   IF "TRUE" THEN
       #_LMDBToDBMZ9(I_CopyDB := #SendAlarm[10],   // "LMDBToDB"
                     I_SourceDB := #C_AlarmDBMZ9,
                     I_StartAddresSourceDB := 0,
                     I_DestDB := #C_AlarmCompareDBMZ9,
                     I_StartAddressDestDB := 0,
                     I_LenghtBytes := #AlarmLength);
   END_IF;
END_REGION

REGION Network 60: **** 5.2 - Flow Equations **** Filter
   // Filter
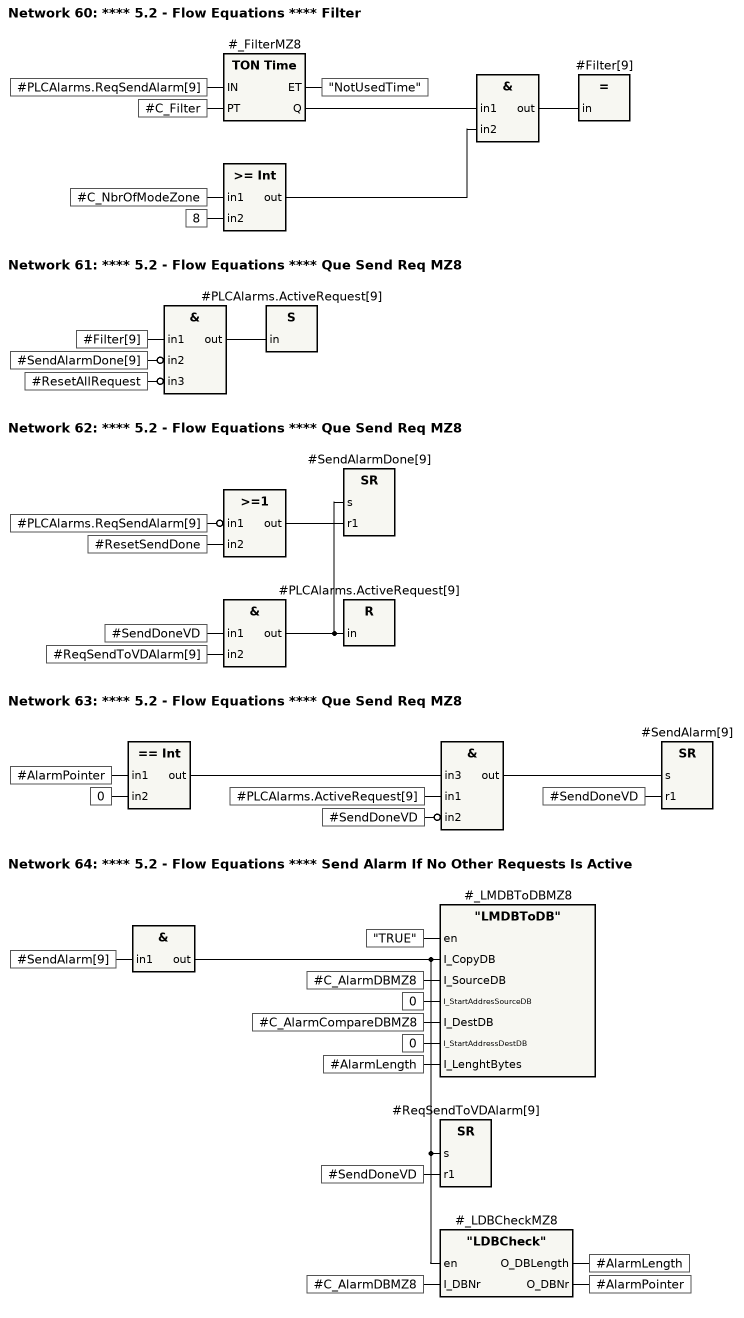
   #_FilterMZ8(IN := #PLCAlarms.ReqSendAlarm[9], PT := #C_Filter, ET => "NotUsedTime");   // TON
   #Filter[9] := #_FilterMZ8.Q AND (#C_NbrOfModeZone >= 8);
END_REGION

REGION Network 61: **** 5.2 - Flow Equations **** Que Send Req MZ8
   // Que Send Req
   IF #Filter[9] AND NOT #SendAlarmDone[9] AND NOT #ResetAllRequest THEN
       #PLCAlarms.ActiveRequest[9] := TRUE;
   END_IF;
END_REGION

REGION Network 62: **** 5.2 - Flow Equations **** Que Send Req MZ8
   // Que Send Req
   #_w1 := #SendDoneVD AND #ReqSendToVDAlarm[9];
   IF #_w1 THEN
       #SendAlarmDone[9] := TRUE;   // SR flip-flop
   END_IF;
   IF NOT #PLCAlarms.ReqSendAlarm[9] OR #ResetSendDone THEN #SendAlarmDone[9] := FALSE; END_IF;
   IF #_w1 THEN #PLCAlarms.ActiveRequest[9] := FALSE; END_IF;
END_REGION

REGION Network 63: **** 5.2 - Flow Equations **** Que Send Req MZ8
   // Que Send Req
   IF (#AlarmPointer = 0) AND #PLCAlarms.ActiveRequest[9] AND NOT #SendDoneVD THEN
       #SendAlarm[9] := TRUE;   // SR flip-flop
   END_IF;
   IF #SendDoneVD THEN #SendAlarm[9] := FALSE; END_IF;
END_REGION

